# B&R Automation Studio project TD52 (part 148)

### Global_DI.var
```iecst
VAR
	VIS2MM : VIS2MM_DI_struct;
	MM2VIS : MM2VIS_DI_struct;
	Para : Para_DI_struct;
	IN_DI : IN_DI_struct;
	OUT_DI : OUT_DI_struct;
	OPC2MM : OPC2MM_DI_struct;
	bComOpcBitTB : BOOL; (*Kommunikation Bit vom Prüfstand über OPC*)
	TON_bComOpcBitTB : TON; (*AliveTime von Opc-Verbindung*)
	TON_bComOpcFailTB : TON; (*Störung Opc-Verbindung*)
	bComOpcBitMDE : BOOL; (*Kommunikation Bit vom Prüfstand über OPC*)
	TON_bComOpcBitMDE : TON; (*AliveTime von Opc-Verbindung MDE*)
	TON_bComOpcFailMDE : TON; (*Störung Opc-Verbindung MDE*)
	rOpcAG_R : ARRAY[0..40] OF REAL; (*REAL-Var zu TB-Control AuxiliariesGeneral*)
	bOpcAG_R : ARRAY[0..30] OF BOOL; (*BOOL-Var zu TB-Control AuxiliariesGeneral*)
	rOpcCU_R : ARRAY[0..50] OF REAL; (*REAL-Var zu TB-Control Customized*)
	rOpcEX_R : ARRAY[0..30] OF REAL; (*REAL-Var zu TB-Control Exhaust*)
	bOpcEX_R : ARRAY[0..20] OF BOOL; (*BOOL-Var zu TB-Control Exhaust*)
	rOpcGT_R : ARRAY[0..50] OF REAL; (*REAL-Var zu TB-Control Gastrain*)
	bOpcGT_R : ARRAY[0..50] OF BOOL; (*BOOL-Var zu TB-Control Gastrain*)
	rOpcHC_R : ARRAY[0..150] OF REAL; (*REAL-Var zu TB-Control HeatingCooling*)
	bOpcHC_R : ARRAY[0..150] OF BOOL; (*BOOL-Var zu TB-Control HeatingCooling*)
	rOpcME_R : ARRAY[0..10] OF REAL; (*REAL-Var zu TB-Control Measurement*)
	bOpcME_R : ARRAY[0..10] OF BOOL; (*BOOL-Var zu TB-Control Measurement*)
	rOpcVE_R : ARRAY[0..50] OF REAL; (*REAL-Var zu TB-Control Ventilation*)
	bOpcVE_R : ARRAY[0..50] OF BOOL; (*BOOL-Var zu TB-Control Ventilation*)
	bOpcMsg_W : ARRAY[0..799] OF BOOL; (*BOOL-Var von TB-Control Message*)
	rOpcAG_W : ARRAY[0..20] OF REAL; (*REAL-Var von TB-Control AuxiliariesGeneral*)
	bOpcAG_W : ARRAY[0..20] OF BOOL; (*BOOL-Var von TB-Control AuxiliariesGeneral*)
	rOpcCU_W : ARRAY[0..50] OF REAL; (*REAL-Var zu TB-Control Customized*)
	rOpcEX_W : ARRAY[0..30] OF REAL; (*REAL-Var von TB-Control Exhaust*)
	bOpcEX_W : ARRAY[0..20] OF BOOL; (*BOOL-Var von TB-Control Exhaust*)
	rOpcGT_W : ARRAY[0..300] OF REAL; (*REAL-Var von TB-Control Gastrain*)
	bOpcGT_W : ARRAY[0..70] OF BOOL; (*BOOL-Var von TB-Control Gastrain*)
	rOpcHC_W : ARRAY[0..380] OF REAL; (*REAL-Var von TB-Control HeatingCooling*)
	bOpcHC_W : ARRAY[0..300] OF BOOL; (*BOOL-Var von TB-Control HeatingCooling*)
	rOpcME_W : ARRAY[0..50] OF REAL; (*REAL-Var von TB-Control Measurement*)
	bOpcME_W : ARRAY[0..20] OF BOOL; (*BOOL-Var von TB-Control Measurement*)
	rOpcVE_W : ARRAY[0..80] OF REAL; (*REAL-Var von TB-Control Ventilation*)
	bOpcVE_W : ARRAY[0..40] OF BOOL; (*BOOL-Var von TB-Control Ventilation*)
	rOpcMDE_R : ARRAY[0..440] OF REAL; (*REAL-Var zu TB-Control Measurement 10ms*)
	bOpcMDE_R : ARRAY[0..20] OF BOOL; (*BOOL-Var zu TB-Control Measurement 10ms*)
	rOpcMDE_W : ARRAY[0..50] OF REAL; (*REAL-Var von TB-Control Measurement 10ms*)
	bOpcMDE_W : ARRAY[0..40] OF BOOL; (*BOOL-Var von TB-Control Measurement 10ms*)
	rGC_CurrentMonth : REAL; (*GC momentaner Monat*)
	rGC_CurrentDay : REAL; (*GC momentaner Tag*)
	rGC_CurrentYear : REAL; (*GC momentanes Jahr*)
	rGC_CurrentHour : REAL; (*GC momentane Stunde*)
	rGC_CurrentMinute : REAL; (*GC momentane Minute*)
	rGC_SampleMonth : REAL; (*GC Probe gezogen Monat*)
	rGC_SampleDay : REAL; (*GC Probe gezogen Tag*)
	rGC_SampleYear : REAL; (*GC Probe gezogen Jahr*)
	rGC_SampleHour : REAL; (*GC Probe gezogen Stunde*)
	rGC_SampleMinute : REAL; (*GC Probe gezogen Minute*)
	TON_DemDataMan_GC : TON; (*Damit der Visu-Button wieder auf FALSE geschrieben wird*)
	rEndurTestTimeMinute : REAL; (*Dauerlauf beendet Tagesminute*)
	rEndurTestTimeHour : REAL; (*Dauerlauf beendet Tagesstunde*)
	rEndurTestTimeDay : REAL; (*Dauerlauf beendet Tag vom Monat*)
	rEndurTestTimeWDay : REAL; (*Dauerlauf beendet Wochentag*)
	rEndurTestTimeMonth : REAL; (*Dauerlauf beendet Monat*)
	rEndurTestTimeYear : REAL; (*Dauerlauf beendet Jahr*)
	rP_MDE_OPC_Set : REAL; (*Externe Leistungsvorgabe von Messtechnik*)
	bMDEBusAlive : BOOL; (*Bus-Verbindung vorhanden für Leistungsvorgabe von Messtechnik*)
	bMDEOPC_Dem : BOOL; (*Anforderung externe Leistungsvorgabe von Messtechnik*)
	RS_Ctr_ChCW_LT : RS; (*Aktivierung Y_Set für Offset*)
	RS_Ctr_ChCW_HT : RS; (*Aktivierung Y_Set für Offset*)
	RS_Ctr_ChCW_LT_LP : RS; (*Aktivierung Y_Set für Offset*)
	RS_Ctr_ChCW_LT_HP : RS; (*Aktivierung Y_Set für Offset*)
	RS_Ctr_ChCW_HT_LP : RS; (*Aktivierung Y_Set für Offset*)
	RS_Ctr_ChCW_HT_HP : RS; (*Aktivierung Y_Set für Offset*)
	RS_Ctr_ECW : RS; (*Aktivierung Y_Set für Offset*)
	RS_Ctr_OCW : RS; (*Aktivierung Y_Set für Offset*)
	bCtr_LT_In_Y_set_Active : BOOL; (*Y_Set für Offset aktiv*)
	bCtr_HT_In_Y_set_Active : BOOL; (*Y_Set für Offset aktiv*)
	bCtr_LT_LP_In_Y_set_Active : BOOL; (*Y_Set für Offset aktiv*)
	bCtr_LT_HP_In_Y_set_Active : BOOL; (*Y_Set für Offset aktiv*)
	bCtr_HT_LP_In_Y_set_Active : BOOL; (*Y_Set für Offset aktiv*)
	bCtr_HT_HP_In_Y_set_Active : BOOL; (*Y_Set für Offset aktiv*)
	bCtr_ECW_In_Y_set_Active : BOOL; (*Y_Set für Offset aktiv*)
	bCtr_OCW_In_Y_set_Active : BOOL; (*Y_Set für Offset aktiv*)
	bBlock_MG_TB : BOOL; (*Block mixgas controller from TB CPU*)
	bBlock_SG_TB : BOOL; (*Block special gas from TB CPU*)
	bDem_GT3 : BOOL; (*activation bit for custom gastrain 3*)
	rGT_RatioAdd : REAL; (*add mixing setpoint for custom gastrain 3*)
	rH2_Set : REAL; (*setpoint addmixing H2*)
	rH2_Act_Calc : REAL; (*Actual volume H2 content calculated (gas meter)*)
	rH2_Act_Cube : REAL; (*Actual volume H2 content measurement cube*)
	rTB_Version : REAL; (*Gesendete Version von TB_Control*)
	bPreHeatWDayLT_On : BOOL; (*Einschalten der Vorwärmung über Zeitsteuerung*)
	usDurationPI_A : UINT := 0; (*PI Duration Bank A*)
	usDurationPI_B : UINT := 0; (*PI Duration Bank B*)
END_VAR
```

### Data object Logical/DataInterface/META_DI (Simple) - Simple data object.

#### META_DI.dat
```
; *******************************************************************************
; AGGR: Module Meta Data (data module)
;
; This code is confidential and proprietary to the INNIO Company.
; It may not be used in any form, or reproduced in any manner, without the express
; written permission of the INNIO Company.
; Copyright, INNIO Company, 2022
;
; Customized modifications: -
; ------------------------
;
; History:
; -------
; V1.00.0	14.11.2022	Vockenberger	Neu erstellt
;
; Instructions for use:
; --------------------
; make only changes at the version numbers
;
; Outstandings:
; ------------
;
; *******************************************************************************
;
"<META>"
;
; Module ID
"<MODUL>DI</MODUL>"
;
; Module Version (xx.yy.zz.cc)
"<VERSION>01.01.00.00</VERSION>"
;
; Module Basisupdate Version BU (00-99)
"<BASISUPDATE_VERSION>00</BASISUPDATE_VERSION>"
;
; Optional: specify order number for limitated module usage
"<ORDER></ORDER>" ;<!--(optional for restricted customizations; missing statement makes module valid for all orders)-->
;
; Permanent Datamodule Filenames<!-- NAME ist ohne Dateiendung einzutragen; Nur für Counter und interne Parameter verwenden-->
"<DATAMODULES>" ;<!-- optional; mehrere DATAMODULES erlaubt-->
"	<DATAMODULE>perm_DI</DATAMODULE>"
"	<DATAMODULE>VISpm_DI</DATAMODULE>"
"</DATAMODULES>"
;
"</META>"
```

### Program Logical/DataInterface/Gnl_AG (IEC) - General Var edit

#### Gnl_AG.st
```iecst
(*******************************************************************************
Gnl_AG		Allgemeine Verarbeitung von Variablen

This code is confidential AND proprietary to the INNIO Company.
It may NOT be used in any form, or reproduced in any manner, without the express
written permission of the INNIO Company.
Copyright, INNIO Company, 2022

Customized modifications: -
------------------------

History:
-------
V1.00.0	14.09.2022		Vockenberger	Neu erstellt
V1.01.0	31.05.2023		Vockenberger	Gaskompressor mit Parameterabfrage und Betriebsstundenzähler mit Wartungsanforderung
										Dauerlauftest
		11.07.2023		Gruber St.		Hinzugefügt: Gasventil 3, Parameter & Anzeigen Gastrain, diverse Abfragen für Visu
		31.07.2023		Vockenberger	Struktur von General_DI geändert
V1.02.0 20.03.2024		Vockenberger	Parameter für Visu Aktivierungen hinzugefügt
		11.04.2024		Vockenberger	Version von 1.01.0 auf 1.02.0 erhöht
V1.02.1 16.10.2024		Vockenberger	Version 1.02.1
V1.03.0	09.01.2025		Gruber St.		cleanUp after change of parameter structure

Instructions FOR use:
--------------------

Outstandings:
------------

*******************************************************************************)

PROGRAM _CYCLIC

	(*DataInterface Version auf Visu Übertragen*)
	MM2VIS.stDI_Version := '1.03.5';

	(*TB_Control Version auf Visu Übertragen*)
	stTB_Version := REAL_TO_STRING(rTB_Version);
	stTB_VersionConfig1 := INSERT(stTB_Version, '.', 1);
	stTB_VersionConfig2 := INSERT(stTB_VersionConfig1, '.', 4);
	strcpy( ADR(MM2VIS.stTB_Version), ADR(stTB_VersionConfig2) );

	(* Parameter für Visu Aktivierungen *)
	Para.bExtCtrNOX_Active;

	(* Zeitsteuerung von Vorwärmung wird Deaktiverit *)
	FOR i:= 0 TO 6 DO
		IF VIS2MM.bECW_PreH_Dem_Customized THEN (*Wenn die Vorwärmung auf der Visu deaktiviert wird, wird die Zeitsteurung auch unterbrochen, bis zum nächsten aktivierten Tag*)
			Para.tPreHeatWDay[i].Off := TRUE;
		ELSE
			Para.tPreHeatWDay[i].Off := FALSE;
		END_IF
	END_FOR

	(* Oil level umrechnen auf % damit der Tank die Füllmenge richtig anzeigt *)
	IF MM2VIS.rLevel_Oiltank > Para.rLevel_Oiltank_ScalY1 AND (Para.rLevel_Oiltank_ScalY2 > 0.0) THEN
		MM2VIS.rLevel_OilNorm := MM2VIS.rLevel_Oiltank/Para.rLevel_Oiltank_ScalY2 *100;
	ELSE
		MM2VIS.rLevel_OilNorm := 0;
	END_IF

	(* Dauerlauftest *)
	DT_EndurTest.minute := REAL_TO_USINT(rEndurTestTimeMinute);
	DT_EndurTest.hour := REAL_TO_USINT(rEndurTestTimeHour);
	DT_EndurTest.day := REAL_TO_USINT(rEndurTestTimeDay);
	DT_EndurTest.wday := REAL_TO_USINT(rEndurTestTimeWDay);
	DT_EndurTest.month := REAL_TO_USINT(rEndurTestTimeMonth);
	DT_EndurTest.year := REAL_TO_UINT(rEndurTestTimeYear);

	ascDTStructure(ADR(DT_EndurTest),ADR(stEndurTestAll),25);
	stFind := ':'; //Es wird nach : gesucht
	iPosition := FIND(stEndurTestAll, stFind);
	szResultString := DELETE(stEndurTestAll, 15, iPosition+3); //Wenn : gefunden wurde, die Position + 3 damit die Position, ab der gelöscht werden soll bestimmt wird
	szDateString := LEFT(szResultString, 10);
	szTimeString := RIGHT(szResultString, 5);

	strcpy( ADR(MM2VIS.stEndurTestDate), ADR(szDateString) );
	strcpy( ADR(MM2VIS.stEndurTestTime), ADR(szTimeString) );

	IF EDGEPOS(MM2VIS.bEndurTestEnd) THEN
		VIS2MM.bEndurTestStart := FALSE; //Start Schalter wird auf False geschrieben, wenn der Test beendet ist
	END_IF

	(*Visu-Button Lüftung auf Automatik wird bei Anfoderung HBT auf TRUE geschrieben*)
	IF IN_DI.bEng_Run OR EDGEPOS(IN_DI.bEng_Aux_Dem_CDR) THEN
		VIS2MM.bDem_ERV_Aut_Vis := TRUE;
	END_IF

	(*Service Page Variablen, nur vorbereitet, keine Funktion*)
	VIS2MM.bManCircLouActive;
	VIS2MM.bManCircLouEngActive;
	VIS2MM.bManDem_PCG_Val;
	VIS2MM.bManFV_PCGC_MG;
	VIS2MM.bManGV_Active;
	VIS2MM.bManGV_NG_Set;
	VIS2MM.bManGV_PG_Set;
	VIS2MM.bManGV_SG_Set;
	VIS2MM.bManInAirFanActive;
	VIS2MM.bManInEngAirFanActive;
	VIS2MM.bManInlLouActive;
	VIS2MM.bManInlLouEngActive;
	VIS2MM.bManInlLouRoomActive;
	VIS2MM.bManOutAirFanActive;
	VIS2MM.bManOutlLouActive;
	VIS2MM.bManPCG_Comp_Active;
	VIS2MM.bManPCG_DemCoolFan;
	VIS2MM.bManPCG_DemReliefValve;
	VIS2MM.bManPCG_DemValCW;
	VIS2MM.bManPCG_GC_Dem;
	VIS2MM.bManPCG_GV_MG_Set;
	VIS2MM.bManPCG_GV_NG_Set;
	VIS2MM.bManPCG_GV_PG_Set;
	VIS2MM.rManCircLouEngSet;
	VIS2MM.rManCircLouSet;
	VIS2MM.rManInAirFanSet;
	VIS2MM.rManInEngAirFanSet;
	VIS2MM.rManInlLouEngSet;
	VIS2MM.rManInlLouRoomSet;
	VIS2MM.rManInlLouSet;
	VIS2MM.rManOutAirFanSet;
	VIS2MM.rManOutlLouSet;

END_PROGRAM
```

#### Gnl_AG.var
```iecst
VAR
	i : INT;
	DT_EndurTest : DTStructure; (*Date and Time Struktur zu weiter Verarbeitung*)
	stFind : STRING[10]; (*Das was im String gesucht wird*)
	stEndurTestAll : STRING[25]; (*Dauerlauftest Datum ganzer String*)
	iPosition : INT; (*Position von : im String*)
	szResultString : STRING[25]; (*Bearbeiteter String*)
	szDateString : STRING[11]; (*Bearbeiteter String, der auf die Visu geschrieben werden kann*)
	szTimeString : STRING[6]; (*Bearbeiteter String, der auf die Visu geschrieben werden kann*)
	stTB_Version : STRING[10]; (*Versionsanzeige TB_Control von REAL auf STRING umgewandelt*)
	stTB_VersionConfig1 : STRING[10]; (*Für TB_Control Versionsanzeige wird der reste Punkt eingefügt*)
	stTB_VersionConfig2 : STRING[6]; (*Für TB_Control Versionsanzeige wird der zweite Punkt eingefügt*)
END_VAR
```

### Program Logical/DataInterface/Gnl_GT (IEC) - General Var edit

#### Gnl_GT.st
```iecst
(*******************************************************************************
Gnl_GT		Allgemeine Verarbeitung von Variablen

This code is confidential AND proprietary to the INNIO Company.
It may NOT be used in any form, or reproduced in any manner, without the express
written permission of the INNIO Company.
Copyright, INNIO Company, 2022

- list addidtional customized IO channels

Customized modifications: -
------------------------

History:
-------
V1.00.0	14.09.2022		Vockenberger	Neu erstellt
V1.01.0	31.05.2023		Vockenberger	Gaskompressor mit Parameterabfrage und Betriebsstundenzähler mit Wartungsanforderung
										Dauerlauftest
										Externe Leistungsvorgabe, umschaltung von Prüfstand/PUMA auf EnergyManagement
		11.07.2023		Gruber St.		Hinzugefügt: Gasventil 3, Parameter & Anzeigen Gastrain, diverse Abfragen für Visu
		31.07.2023		Vockenberger	Struktur von General_DI geändert
		09.01.2024		Gruber St.		added blockage bits for mixgas & special gas
V1.01.1	19.03.2024		Gruber St.		added vis mixgas ratio from IN_DI
		27.03.2024		Gruber St.		added vis H2 measurement cube
V1.02.0	22.04.2024		Gruber St.		Parameter for several vis; MFC open vis
V1.03.0	14.01.2025		Gruber St.		several changes for new para struct

Instructions FOR use:
--------------------

Outstandings:
------------

*******************************************************************************)

PROGRAM _CYCLIC

	(* ----------------------------------------------------------------------------*)
	(*Uhrzeit vom GC generieren*)
	iGC_CurrentDay := REAL_TO_SINT(rGC_CurrentDay);
	iGC_CurrentMonth := REAL_TO_USINT(rGC_CurrentMonth);
	iGC_CurrentYear := REAL_TO_UINT(rGC_CurrentYear);
	iGC_CurrentHour := REAL_TO_USINT(rGC_CurrentHour);
	iGC_CurrentMinute := REAL_TO_USINT(rGC_CurrentMinute);

	iGC_SampleDay := REAL_TO_SINT(rGC_SampleDay);
	iGC_SampleMonth := REAL_TO_USINT(rGC_SampleMonth);
	iGC_SampleYear := REAL_TO_UINT(rGC_SampleYear);
	iGC_SampleHour := REAL_TO_USINT(rGC_SampleHour);
	iGC_SampleMinute := REAL_TO_USINT(rGC_SampleMinute);

	GC_CurrentDate.day := iGC_CurrentDay;
	GC_CurrentDate.month := iGC_CurrentMonth;
	GC_CurrentDate.year := iGC_CurrentYear;

	GC_CurrentTIME.hour := iGC_CurrentHour;
	GC_CurrentTIME.minute := iGC_CurrentMinute;

	GC_SampleDate.day := iGC_SampleDay;
	GC_SampleDate.month := iGC_SampleMonth;
	GC_SampleDate.year := iGC_SampleYear;

	GC_SampleTIME.hour := iGC_SampleHour;
	GC_SampleTIME.minute := iGC_SampleMinute;

	LenTime:=6;
	LenDate:=25;
	ascDTStructure(ADR(GC_CurrentDate),ADR(MM2VIS.stGC_CurrentDate),LenDate);  (* converts TIMEStructure to a string *)
	ascTIMEStructure(ADR(GC_CurrentTIME),ADR(MM2VIS.stGC_CurrentTIME),LenTime);

	ascDTStructure(ADR(GC_SampleDate),ADR(MM2VIS.stGC_SampleDate),LenDate);
	ascTIMEStructure(ADR(GC_SampleTIME),ADR(MM2VIS.stGC_SampleTIME),LenTime);

	(* ----------------------------------------------------------------------------*)
	(* Visualization mixgas ratio *)
	IF Para.bGasFlowCtr AND NOT Para.bIncl_SG_Calc OR (NOT Para.bGasFlowCtr AND NOT Para.bIncl_SG_Calc) THEN
		MM2VIS.rVol_NG_PG := MM2VIS.rVol_NG + MM2VIS.rVol_PG - MM2VIS.rVol_SG;
	ELSE
		MM2VIS.rVol_NG_PG := MM2VIS.rVol_NG + MM2VIS.rVol_PG; (* part of special gas already included *)
	END_IF;

	(* Visualization MFC propan gas open *)
	IF MM2VIS.rCtr_MFC_PG > 0.01 THEN
		MM2VIS.bMFC_PG_open_vis := TRUE;
	ELSE
		MM2VIS.bMFC_PG_open_vis := FALSE;
	END_IF;

	(* Visualization MFC special gas open *)
	IF MM2VIS.rCtr_MFC_SG > 0.01 THEN
		MM2VIS.bMFC_SG_open_vis := TRUE;
	ELSE
		MM2VIS.bMFC_SG_open_vis := FALSE;
	END_IF;

	(* Visualization H2 measurement cube *)
	MM2VIS.rH2_Act_Cube	:= rH2_Act_Cube * 100;

	(* Abfrage für Freigabe Mischgas-Regler mittels Gasdosierventil - Gas 1-2/3 *)
	IF IN_DI.iIdx_Gastyp = 3
		AND IN_DI.iNum_GT = 2
		AND IN_DI.bTJ_Exist = TRUE
		AND IN_DI.iN_GMU_Devices > 1
		AND IN_DI.bGT_MixActive = TRUE
		AND (IN_DI.iIdx_SelGasTyp = 6 OR IN_DI.iIdx_SelGasTyp = 5)
		AND MM2VIS.bDem_GV_PG
		AND NOT MM2VIS.bDem_GV_SG THEN
		MM2VIS.bParaGasMixEngOk := TRUE;
	ELSE
		MM2VIS.bParaGasMixEngOk := FALSE;
	END_IF;

	(* Abfrage für Freigabe Mischgas-Regler mittels MFC - Gas 1-2 *)
	IF IN_DI.iIdx_Gastyp >= 2
		AND IN_DI.iIdx_SelGasTyp = 0
		AND IN_DI.bGT_CVActive
		AND IN_DI.bGT_CVIpol12Active THEN
		MM2VIS.bParaGasMixMFCOk := TRUE;
	ELSE
		MM2VIS.bParaGasMixMFCOk := FALSE;
	END_IF

	(* Freigabe Mischgas für Anzeige auf Visu *)
	IF MM2VIS.bParaGasMixMFCOk OR MM2VIS.bParaGasMixEngOk THEN
		MM2VIS.bRelMixGas := TRUE;
	ELSE
		MM2VIS.bRelMixGas := FALSE;
	END_IF;

	(* Switch Mixgas from MN-Controller to Volume - Gas 1-2 *)
	IF EDGENEG(MM2VIS.bParaGasMixMFCOk AND NOT (MM2VIS.bDem_GV_NG AND MM2VIS.bDem_GV_PG AND MM2VIS.bDem_GV_SG AND Para.bIncl_SG_Calc)) AND VIS2MM.bCtr_MN_MG_active THEN
		VIS2MM.bVolPG_Man := TRUE;
	END_IF;

	(* Switch Mixgas from MN-Controller to Off - Gas 1-2/3 *)
	IF EDGENEG(MM2VIS.bParaGasMixEngOk AND NOT (MM2VIS.bDem_GV_NG AND MM2VIS.bDem_GV_PG AND MM2VIS.bDem_GV_SG AND Para.bIncl_SG_Calc)) AND VIS2MM.bCtr_MN_MG_active THEN
		VIS2MM.bCtr_MN_MG_off := TRUE;
	END_IF;

	(* Block mixgas controller *)
	IF bBlock_MG_TB OR MM2VIS.bMsg7000 THEN
		VIS2MM.bCtr_MN_MG_off := TRUE;
	END_IF;

	(* Block specialgas mixing *)
	IF bBlock_SG_TB OR MM2VIS.bMsg7000 THEN
		VIS2MM.rVol_SG_Set := 0;
	END_IF;

	(* Externe Anforderung MZ von PUMA *)
	IF VIS2MM.bExtMN_ActiveMDE AND MM2VIS.bExtMNFromMDE THEN
		VIS2MM.bCtr_MN_MG_active := TRUE;
		Para.tCtr_MN_MG.W_set := MM2VIS.rExtMN_Set;
	END_IF;

	IF EDGENEG(VIS2MM.bExtMN_ActiveMDE) THEN
		VIS2MM.bCtr_MN_MG_off := TRUE;
	END_IF;

	(* Switch Mixgas from Volume to OFF *)
	IF EDGENEG(MM2VIS.bParaGasMixMFCOk OR (MM2VIS.bDem_GV_NG AND MM2VIS.bDem_GV_PG AND MM2VIS.bDem_GV_SG)) AND VIS2MM.bVolPG_Man THEN
		VIS2MM.bCtr_MN_MG_off := TRUE;
	END_IF;

	(* Wenn MN Bechrechnung inaktiv, dann wird der MN-Regler deaktiviert *)
	IF EDGENEG(MM2VIS.bMN_Cal_Status) THEN
		VIS2MM.bCtr_MN_MG_off := TRUE;
	END_IF;

	(* MN Ctr from MN to OFF *)
	IF EDGEPOS(VIS2MM.bCtr_MN_MG_off) AND VIS2MM.bCtr_MN_MG_active THEN
		Para.tCtr_MN_MG.W_set := 100;
	ELSE
		Para.tCtr_MN_MG.W_set := Para.tCtr_MN_MG.W_set;
	END_IF

	(* MN Ctr from Volume to OFF *)
	IF EDGEPOS(VIS2MM.bCtr_MN_MG_off) AND VIS2MM.bVolPG_Man THEN
		VIS2MM.rVol_PG_Set := 0;
	ELSE
		VIS2MM.rVol_PG_Set := VIS2MM.rVol_PG_Set;
	END_IF

	(* MN Ctr from MN to VOL *)
	IF EDGEPOS(VIS2MM.bVolPG_Man) AND VIS2MM.bCtr_MN_MG_active THEN
		VIS2MM.rVol_PG_Set := MM2VIS.rVol_PG;
	ELSE
		VIS2MM.rVol_PG_Set := VIS2MM.rVol_PG_Set;
	END_IF

	(* MN Ctr from VOL to MN *)
	IF EDGEPOS(VIS2MM.bCtr_MN_MG_active) AND VIS2MM.bVolPG_Man THEN
		Para.tCtr_MN_MG.W_set := MM2VIS.rMN_MG;
	ELSE
		Para.tCtr_MN_MG.W_set := Para.tCtr_MN_MG.W_set;
	END_IF

	(* Regler Methane Button Steuerung *)
	 IF EDGEPOS(VIS2MM.bCtr_MN_MG_active) THEN
		VIS2MM.bCtr_MN_MG_off := FALSE;
		VIS2MM.bVolPG_Man := FALSE;
	ELSE
		VIS2MM.bCtr_MN_MG_off := VIS2MM.bCtr_MN_MG_off;
		VIS2MM.bVolPG_Man := VIS2MM.bVolPG_Man;
	END_IF

	IF EDGEPOS(VIS2MM.bCtr_MN_MG_off) THEN
		VIS2MM.bCtr_MN_MG_active := FALSE;
		VIS2MM.bVolPG_Man := FALSE;
	ELSE
		VIS2MM.bCtr_MN_MG_active := VIS2MM.bCtr_MN_MG_active;
		VIS2MM.bVolPG_Man := VIS2MM.bVolPG_Man;
	END_IF

	IF EDGEPOS(VIS2MM.bVolPG_Man) THEN
		VIS2MM.bCtr_MN_MG_active := FALSE;
		VIS2MM.bCtr_MN_MG_off := FALSE;
	ELSE
		VIS2MM.bCtr_MN_MG_active := VIS2MM.bCtr_MN_MG_active;
		VIS2MM.bCtr_MN_MG_off := VIS2MM.bCtr_MN_MG_off;
	END_IF

	IF EDGENEG(MM2VIS.bDem_GV_SG) THEN
		VIS2MM.rVol_SG_Set := 0;
	ELSE
		VIS2MM.rVol_SG_Set := VIS2MM.rVol_SG_Set;
	END_IF

	(* ----------------------------------------------------------------------------*)
	(* Gaskompressor Wartungsanforderung *)
	IF Para.bGasCompActive THEN
		xComp_OpHour(enable := MM2VIS.bPr_PCG_GC_Dem, BH_adr := ADR(ComOpHour_Imp.tick));
		xTOF_CompOpHour(IN := xComp_OpHour.BH_Imp, PT := T#10s);
		IF EDGEPOS(xTOF_CompOpHour.Q) THEN
			Para.rCnt_CompOpHoursW := Para.rCnt_CompOpHoursW - 1;					(* increase counter *)
		END_IF
		Para.rCnt_CompOpHoursW 			:= Para.rCnt_CompOpHoursW;

		IF Para.rCnt_CompOpHoursW <= 0 THEN
			OUT_DI.bCompOpHoursWarning := TRUE;
		ELSE
			OUT_DI.bCompOpHoursWarning := FALSE;
		END_IF
	END_IF

	(* ----------------------------------------------------------------------------*)
	(* set PG trace heating on, with time control *)
	IF EDGEPOS(MM2VIS.bPG_TraceHeat_TimeCtr_On) THEN
		VIS2MM.bSel_PG_TraceHeat := TRUE;
	END_IF

	(* ----------------------------------------------------------------------------*)
	(* Added Parameter bSA_PI_Active AND to TB_Control-VIS *)
	MM2VIS.bSA_PI_Active := IN_DI.bSA_PI_Active;
	MM2VIS.rCA_PI_Dur_Avg := IN_DI.rCA_PI_Dur_Avg;

END_PROGRAM
```

#### Gnl_GT.var
```iecst
VAR
	iGC_CurrentDay : USINT; (*GC momentaner Tag*)
	iGC_CurrentMonth : USINT; (*GC momentaner Monat*)
	iGC_CurrentYear : UINT; (*GC momentanes Jahr*)
	iGC_CurrentHour : USINT; (*GC momentane Stunde*)
	iGC_CurrentMinute : USINT; (*GC momentane Minute*)
	iGC_SampleDay : USINT; (*GC Probe gezogen Tag*)
	iGC_SampleMonth : USINT; (*GC Probe gezogen Monat*)
	iGC_SampleYear : UINT; (*GC Probe gezogen Jahr*)
	iGC_SampleHour : USINT; (*GC Probe gezogen Stunde*)
	iGC_SampleMinute : USINT; (*GC Probe gezogen Minute*)
	GC_SampleTIME : TIMEStructure; (*GC TimeStructure für VisuString*)
	GC_CurrentTIME : TIMEStructure; (*GC TimeStructure für VisuString*)
	GC_SampleDate : DTStructure; (*GC DateStructure für VisuString*)
	GC_CurrentDate : DTStructure; (*GC DateStructure für VisuString*)
	LenTime : UDINT; (*GC VisuString-Länge für Anzeige*)
	LenDate : UDINT; (*GC VisuString-Länge für Anzeige*)
	ComOpHour_Imp : bh_typ; (*Compressor operation hours counter*)
	xComp_OpHour : BH; (*Hour counter for compressor operating hours*)
	xTOF_CompOpHour : TOF; (*Off delay for compressor operating hours*)
END_VAR
```

### Program Logical/DataInterface/Gnl_HC (IEC) - General Var edit

#### Gnl_HC.st
```iecst
(*******************************************************************************
Gnl_HC		Allgemeine Verarbeitung von Variablen

This code is confidential AND proprietary to the INNIO Company.
It may NOT be used in any form, or reproduced in any manner, without the express
written permission of the INNIO Company.
Copyright, INNIO Company, 2023

- list addidtional customized IO channels

Customized modifications: -
------------------------

History:
-------
V1.01.0	27.05.2023		Vockenberger	Manuelle Anforderung der Kühlkreispumpen, wenn BWS auf Aus ist.
		31.07.2023		Vockenberger	Struktur von General_DI geändert
		09.10.2023		Vockenberger	Offset für Kühlkreis-Regelventile bei Eng_Run eingefügt

Instructions FOR use:
--------------------

Outstandings:
------------

*******************************************************************************)

PROGRAM _CYCLIC

	(* Manuelle Anforderung der Kühlwasserpumpen, wenn Betriebswahlschalter auf aus ist *)
	MM2VIS.iIdx_OMSS := IN_DI.iIdx_OMSS;	//Damit auf der Visualisierung die Schalter verreigelt werden können
	IF IN_DI.iIdx_OMSS = 0 AND NOT IN_DI.bEng_Aux_Dem_CDR THEN
		VIS2MM.bMan_ECW_Pump;
		VIS2MM.bMan_OCW_Pump;
		VIS2MM.bMan_LT_Pump;
		VIS2MM.bMan_HT_Pump;
		VIS2MM.bMan_LT_LP_Pump;
		VIS2MM.bMan_LT_HP_Pump;
		VIS2MM.bMan_HT_LP_Pump;
		VIS2MM.bMan_HT_HP_Pump;
	ELSE
		VIS2MM.bMan_ECW_Pump := FALSE;
		VIS2MM.bMan_OCW_Pump := FALSE;
		VIS2MM.bMan_LT_Pump := FALSE;
		VIS2MM.bMan_HT_Pump := FALSE;
		VIS2MM.bMan_LT_LP_Pump := FALSE;
		VIS2MM.bMan_LT_HP_Pump := FALSE;
		VIS2MM.bMan_HT_LP_Pump := FALSE;
		VIS2MM.bMan_HT_HP_Pump := FALSE;
	END_IF

	(*Aktivierung Offset für Kühlkreis-Regelventile bei Eng_Run*)
	RS_Ctr_ChCW_LT(SET:=EDGEPOS(IN_DI.bEng_Run), RESET1:=(VIS2MM.tCtr_ChCW_LT_In.Y_set < MM2VIS.tCtr_ChCW_LT_Out.Y) OR (EDGENEG(IN_DI.bEng_Run)));
	IF VIS2MM.tCtr_ChCW_LT_In.Y_set_Active AND RS_Ctr_ChCW_LT.Q1 THEN
		bCtr_LT_In_Y_set_Active :=  TRUE;
	ELSE
		bCtr_LT_In_Y_set_Active :=  FALSE;
	END_IF

	RS_Ctr_ChCW_HT(SET:=EDGEPOS(IN_DI.bEng_Run), RESET1:=(VIS2MM.tCtr_ChCW_HT_In.Y_set < MM2VIS.tCtr_ChCW_HT_Out.Y) OR (EDGENEG(IN_DI.bEng_Run)));
	IF VIS2MM.tCtr_ChCW_HT_In.Y_set_Active AND RS_Ctr_ChCW_HT.Q1 THEN
		bCtr_HT_In_Y_set_Active :=  TRUE;
	ELSE
		bCtr_HT_In_Y_set_Active :=  FALSE;
	END_IF

	RS_Ctr_ChCW_LT_LP(SET:=EDGEPOS(IN_DI.bEng_Run), RESET1:=(VIS2MM.tCtr_ChCW_LT_LP_In.Y_set < MM2VIS.tCtr_ChCW_LT_LP_Out.Y) OR (EDGENEG(IN_DI.bEng_Run)));
	IF VIS2MM.tCtr_ChCW_LT_LP_In.Y_set_Active AND RS_Ctr_ChCW_LT_LP.Q1 THEN
		bCtr_LT_LP_In_Y_set_Active :=  TRUE;
	ELSE
		bCtr_LT_LP_In_Y_set_Active :=  FALSE;
	END_IF

	RS_Ctr_ChCW_LT_HP(SET:=EDGEPOS(IN_DI.bEng_Run), RESET1:=(VIS2MM.tCtr_ChCW_LT_HP_In.Y_set < MM2VIS.tCtr_ChCW_LT_HP_Out.Y) OR (EDGENEG(IN_DI.bEng_Run)));
	IF VIS2MM.tCtr_ChCW_LT_HP_In.Y_set_Active AND RS_Ctr_ChCW_LT_HP.Q1 THEN
		bCtr_LT_HP_In_Y_set_Active :=  TRUE;
	ELSE
		bCtr_LT_HP_In_Y_set_Active :=  FALSE;
	END_IF

	RS_Ctr_ChCW_HT_LP(SET:=EDGEPOS(IN_DI.bEng_Run), RESET1:=(VIS2MM.tCtr_ChCW_HT_LP_In.Y_set < MM2VIS.tCtr_ChCW_HT_LP_Out.Y) OR (EDGENEG(IN_DI.bEng_Run)));
	IF VIS2MM.tCtr_ChCW_HT_LP_In.Y_set_Active AND RS_Ctr_ChCW_HT_LP.Q1 THEN
		bCtr_HT_LP_In_Y_set_Active :=  TRUE;
	ELSE
		bCtr_HT_LP_In_Y_set_Active :=  FALSE;
	END_IF

	RS_Ctr_ChCW_HT_HP(SET:=EDGEPOS(IN_DI.bEng_Run), RESET1:=(VIS2MM.tCtr_ChCW_HT_HP_In.Y_set < MM2VIS.tCtr_ChCW_HT_HP_Out.Y) OR (EDGENEG(IN_DI.bEng_Run)));
	IF VIS2MM.tCtr_ChCW_HT_HP_In.Y_set_Active AND RS_Ctr_ChCW_HT_HP.Q1 THEN
		bCtr_HT_HP_In_Y_set_Active :=  TRUE;
	ELSE
		bCtr_HT_HP_In_Y_set_Active :=  FALSE;
	END_IF

	RS_Ctr_ECW(SET:=EDGEPOS(IN_DI.bEng_Run), RESET1:=(VIS2MM.tCtr_ECW_In.Y_set < MM2VIS.tCtr_ECW_Out.Y) OR (EDGENEG(IN_DI.bEng_Run)));
	IF VIS2MM.tCtr_ECW_In.Y_set_Active AND RS_Ctr_ECW.Q1 THEN
		bCtr_ECW_In_Y_set_Active :=  TRUE;
	ELSE
		bCtr_ECW_In_Y_set_Active :=  FALSE;
	END_IF

	RS_Ctr_OCW(SET:=EDGEPOS(IN_DI.bEng_Run), RESET1:=(VIS2MM.tCtr_OCW_In.Y_set < MM2VIS.tCtr_OCW_Out.Y) OR (EDGENEG(IN_DI.bEng_Run)));
	IF VIS2MM.tCtr_OCW_In.Y_set_Active AND RS_Ctr_ECW.Q1 THEN
		bCtr_OCW_In_Y_set_Active :=  TRUE;
	ELSE
		bCtr_OCW_In_Y_set_Active :=  FALSE;
	END_IF

	(*Aktivierung NT Vorwärmung, wenn Betriebswahlschalter auf aus ist über Zeitsteuerung*)
	IF EDGEPOS(bPreHeatWDayLT_On) THEN	(*Aktivierung Vorwärmung vom Prüfstand über eine positiven Flanke*)
		VIS2MM.bLT_PreH_Dem := TRUE;
	ELSE
		VIS2MM.bLT_PreH_Dem := VIS2MM.bLT_PreH_Dem;
	END_IF

	(* Zeitsteuerung von NT Vorwärmung wird Deaktiverit *)
	FOR i:= 0 TO 6 DO
		IF VIS2MM.bLT_PreH_Dem THEN (*Wenn die Vorwärmung auf der Visu deaktiviert wird, wird die Zeitsteurung auch unterbrochen, bis zum nächsten aktivierten Tag*)
			VIS2MM.tPreHeatWDayLT[i].Off := TRUE;
		ELSE
			VIS2MM.tPreHeatWDayLT[i].Off := FALSE;
		END_IF
	END_FOR

END_PROGRAM
```

#### Gnl_HC.var
```iecst
VAR
	i : INT;
END_VAR
```

### Program Logical/DataInterface/Gnl_ME (IEC) - General Var edit

#### Gnl_ME.st
```iecst
(*******************************************************************************
Gnl_ME		Allgemeine Verarbeitung von Variablen

This code is confidential AND proprietary to the INNIO Company.
It may NOT be used in any form, or reproduced in any manner, without the express
written permission of the INNIO Company.
Copyright, INNIO Company, 2023

- list addidtional customized IO channels

Customized modifications: -
------------------------

History:
-------
V1.01.0	31.05.2023	Vockenberger	Externe Leistungsvorgabe, umschaltung von Prüfstand/PUMA auf EnergyManagement
		31.07.2023	Vockenberger	Struktur von General_DI geändert
V1.03.0 10.06.2025	Vockenberger	added extern setpoint for CAT temp over MDE

Instructions FOR use:
--------------------

Outstandings:
------------

*******************************************************************************)

PROGRAM _CYCLIC

	(* Externe Leistungsvorgabe, umschaltung von Prüfstand/PUMA auf EnergyManagement *)
	IF VIS2MM.iSelExtP_OPC_Set = 0 THEN //Externe Leistungvorgabe deaktiviert
		MM2VIS.rP_OPC_Set;
		MM2VIS.bBusAlive := bMDEBusAlive;
		MM2VIS.bOPC_Dem := FALSE;
	ELSIF VIS2MM.iSelExtP_OPC_Set = 1 THEN //Externe Leistungvorgabe über MDE
		MM2VIS.rP_OPC_Set	:= rP_MDE_OPC_Set;
		MM2VIS.bBusAlive := bMDEBusAlive;
		MM2VIS.bOPC_Dem := bMDEOPC_Dem;
	ELSIF VIS2MM.iSelExtP_OPC_Set = 2 THEN  //Externe Leistungvorgabe über EnergyManagement
		MM2VIS.rP_OPC_Set := OPC2MM.rP_OPC_Set;
		MM2VIS.bBusAlive := OPC2MM.bBusAlive;
		MM2VIS.bOPC_Dem := OPC2MM.bOPC_Dem;
	END_IF

	IF EDGEPOS(VIS2MM.iSelExtP_OPC_Set = 0) OR EDGEPOS(VIS2MM.iSelExtP_OPC_Set = 1) OR EDGEPOS(VIS2MM.iSelExtP_OPC_Set = 2) THEN //Beim Umschalten der externen Leistungvorgabe,
		MM2VIS.bOPC_Dem := FALSE;																								 //wird der Motor abgefordert, falls die OPC-Verbidnung nicht vorhanden ist
	END_IF

	(*PI Duration A B*)
	usDurationPI_A	:= 0;
	usDurationPI_B	:= 0;
	FOR i:= 1 TO 5 DO
		usDurationPI_A	:= usDurationPI_A + IN_DI.tPIopenL[i].duration 	+ IN_DI.tPIopenH[i].duration;
		usDurationPI_B	:= usDurationPI_B + IN_DI.tPIopenL[i+5].duration + IN_DI.tPIopenH[i+5].duration;
	END_FOR

	(*Ext CAT temp setpoint*)
	MM2VIS.rCAT_TempSet 				:=	IN_DI.rCAT_TempSet;
	MM2VIS.bExtCAT_TempStatus_Active	:=	OUT_DI.bExtCAT_Temp_Active;
	MM2VIS.rExtCAT_TempSet				:=	OUT_DI.rExtCAT_TempSet;

END_PROGRAM
```

#### Gnl_ME.var
```iecst
VAR
	i : INT;
END_VAR
```

### Program Logical/DataInterface/OpcAG (IEC) - OPC Var for Testbench

#### OpcAG.st
```iecst
(*******************************************************************************
OpcAG	 Variables read or write to Testbench

This code is confidential AND proprietary to the INNIO Company.
It may NOT be used in any form, or reproduced in any manner, without the express
written permission of the INNIO Company.
Copyright, INNIO Company, 2022

- list addidtional customized IO channels

Customized modifications: -
------------------------

History:
-------
V1.00.0	14.09.2022		Vockenberger	Neu erstellt
V1.01.0	25.05.2023		Vockenberger	Dauerlauftest hinzugefügt
		28.07.2023		Vockenberger	Struktur von OPC_DI geändert
		01.08.2023		Vockenberger	Parameter für Öltankskalierung hinzugefügt
		11.01.2024		Vockenberger	bEOVal_DemOpen eingefügt
V1.02.0 10.04.2024		Vockenberger	Betriebswahlschalter, Anforderungsschalter und SY-Schalter eingefügt
V1.02.1	30.10.2024		Vockenberger	ParaTB.rTB_Cust von 1..10 auf 1..19 geändert
V1.03.0	09.01.2025		Gruber St.		cleanUp after change of parameter structure

Instructions FOR use:
--------------------

Outstandings:
------------

*******************************************************************************)

PROGRAM _CYCLIC

	(**Wird von Motor-CPU geschrieben**********************)
	(**REAL**)
	rOpcAG_R[0]		:=	Para.tPreHeatWDay[0].Hour;
	rOpcAG_R[1]		:=	Para.tPreHeatWDay[0].Minute;
	rOpcAG_R[2]		:=	Para.tPreHeatWDay[1].Hour;
	rOpcAG_R[3]		:=	Para.tPreHeatWDay[1].Minute;
	rOpcAG_R[4]		:=	Para.tPreHeatWDay[2].Hour;
	rOpcAG_R[5]		:=	Para.tPreHeatWDay[2].Minute;
	rOpcAG_R[6]		:=	Para.tPreHeatWDay[3].Hour;
	rOpcAG_R[7]		:=	Para.tPreHeatWDay[3].Minute;
	rOpcAG_R[8]		:=	Para.tPreHeatWDay[4].Hour;
	rOpcAG_R[9]		:=	Para.tPreHeatWDay[4].Minute;
	rOpcAG_R[10]	:=	Para.tPreHeatWDay[5].Hour;
	rOpcAG_R[11]	:=	Para.tPreHeatWDay[5].Minute;
	rOpcAG_R[12]	:=	Para.tPreHeatWDay[6].Hour;
	rOpcAG_R[13]	:=	Para.tPreHeatWDay[6].Minute;

	rOpcAG_R[14]	:=	VIS2MM.rEndurTestTimeSet;
	rOpcAG_R[15]	:=	IN_DI.rP_Act_Filt;
	rOpcAG_R[16]	:=	INT_TO_REAL(IN_DI.iIdx_OMSS);
	rOpcAG_R[17]	:=	INT_TO_REAL(IN_DI.iIdx_RSS);
	rOpcAG_R[18]	:=	INT_TO_REAL(IN_DI.iIdx_SyOMSS);

	rOpcAG_R[19];
	rOpcAG_R[20];
	rOpcAG_R[21];
	rOpcAG_R[22];
	rOpcAG_R[23];
	rOpcAG_R[24];
	rOpcAG_R[25];
	rOpcAG_R[26];
	rOpcAG_R[27];
	rOpcAG_R[28];
	rOpcAG_R[29];

	rOpcAG_R[30];
	rOpcAG_R[31];
	rOpcAG_R[32];
	rOpcAG_R[33];
	rOpcAG_R[34];
	rOpcAG_R[35];
	rOpcAG_R[36];
	rOpcAG_R[37];
	rOpcAG_R[38];
	rOpcAG_R[39];
	rOpcAG_R[40];

	(**BOOL**)
	IF MM2VIS.bCtrlBatMon_TestRunning THEN //Damit der Visu-Button wieder auf FALSE geschrieben wird
		VIS2MM.bCtrlBatMon_ManTestStart := FALSE;
	END_IF
	bOpcAG_R[0]	:=	VIS2MM.bCtrlBatMon_ManTestStart;
	bOpcAG_R[1]	:=	IN_DI.bImp_Start;
	bOpcAG_R[2]	:=	Para.tPreHeatWDay[0].Active;
	bOpcAG_R[3]	:=	Para.tPreHeatWDay[0].Off;
	bOpcAG_R[4]	:=	Para.tPreHeatWDay[1].Active;
	bOpcAG_R[5]	:=	Para.tPreHeatWDay[1].Off;
	bOpcAG_R[6]	:=	Para.tPreHeatWDay[2].Active;
	bOpcAG_R[7]	:=	Para.tPreHeatWDay[2].Off;
	bOpcAG_R[8]	:=	Para.tPreHeatWDay[3].Active;
	bOpcAG_R[9]	:=	Para.tPreHeatWDay[3].Off;

	bOpcAG_R[10]	:=	Para.tPreHeatWDay[4].Active;
	bOpcAG_R[11]	:=	Para.tPreHeatWDay[4].Off;
	bOpcAG_R[12]	:=	Para.tPreHeatWDay[5].Active;
	bOpcAG_R[13]	:=	Para.tPreHeatWDay[5].Off;
	bOpcAG_R[14]	:=	Para.tPreHeatWDay[6].Active;
	bOpcAG_R[15]	:=	Para.tPreHeatWDay[6].Off;
	bOpcAG_R[16]	:=	Para.bPreHeatWDay_CtrActive;
	bOpcAG_R[17]	:=	VIS2MM.bEndurTestStart;
	bOpcAG_R[18]	:=	IN_DI.bEOVal_DemOpen;
	bOpcAG_R[19];

	bOpcAG_R[20];
	bOpcAG_R[21];
	bOpcAG_R[22];
	bOpcAG_R[23];
	bOpcAG_R[24];
	bOpcAG_R[25];
	bOpcAG_R[26];
	bOpcAG_R[27];
	bOpcAG_R[28];
	bOpcAG_R[29];
	bOpcAG_R[30];

	(*AuxiliariesGeneral from Testbench*)
	(**REAL**)
	MM2VIS.rU_CtrlBat1			:=	rOpcAG_W[0];
	MM2VIS.rU_CtrlBat_BatTest1	:=	rOpcAG_W[1];
	MM2VIS.rLevel_Oiltank		:=	rOpcAG_W[2];
	rEndurTestTimeMinute		:=	rOpcAG_W[3];
	rEndurTestTimeHour			:=	rOpcAG_W[4];
	rEndurTestTimeDay			:=	rOpcAG_W[5];
	rEndurTestTimeWDay			:=	rOpcAG_W[6];
	rEndurTestTimeMonth			:=	rOpcAG_W[7];
	rEndurTestTimeYear			:=	rOpcAG_W[8];
	rTB_Version					:=	rOpcAG_W[9];

	Para.rLevel_Oiltank_ScalY1	:= rOpcAG_W[10];
	Para.rLevel_Oiltank_ScalY2	:= rOpcAG_W[11];
	MM2VIS.rI_Aux				:= rOpcAG_W[12];
	MM2VIS.rP_Aux				:= rOpcAG_W[13];
	rOpcAG_W[14];
	rOpcAG_W[15];
	rOpcAG_W[16];
	rOpcAG_W[17];
	rOpcAG_W[18];
	rOpcAG_W[19];
	rOpcAG_W[20];

	(**BOOL**)
	MM2VIS.bCtrlBatMon_TestRunning	:= bOpcAG_W[0];
	MM2VIS.bReq_RefillOilPuEng		:= bOpcAG_W[1];
	MM2VIS.bDem_RefillOilPuEng		:= bOpcAG_W[2];
	MM2VIS.bPreHeatWDay_On			:= bOpcAG_W[3];
	MM2VIS.bEndurTestEnd			:= bOpcAG_W[4];
	MM2VIS.bRelAux_TB 				:= bOpcAG_W[5];
	Para.bBatCtrActive				:= bOpcAG_W[6];
	MM2VIS.bServicePageActive		:= bOpcAG_W[7];
	MM2VIS.bAirCompressor1_Run		:= bOpcAG_W[8];
	MM2VIS.bAirCompressor2_Run		:= bOpcAG_W[9];

	bOpcAG_W[10];
	bOpcAG_W[11];
	bOpcAG_W[12];
	bOpcAG_W[13];
	bOpcAG_W[14];
	bOpcAG_W[15];
	bOpcAG_W[16];
	bOpcAG_W[17];
	bOpcAG_W[18];
	bOpcAG_W[20];

END_PROGRAM
```

### Program Logical/DataInterface/OpcCU (IEC) - OPC Var for Testbench

#### OpcCU.st
```iecst
(*******************************************************************************
OpcCU	 Variables read or write to Testbench

This code is confidential AND proprietary to the INNIO Company.
It may NOT be used in any form, or reproduced in any manner, without the express
written permission of the INNIO Company.
Copyright, INNIO Company, 2025

- list addidtional customized IO channels

Customized modifications: -
------------------------

History:
-------
V1.03.0 22.01.2025	Gruber St.	new created

Instructions FOR use:
--------------------

Outstandings:
------------

*******************************************************************************)

PROGRAM _CYCLIC

	(*------------------------------------------------------------------------------
								Testbench to Engine
	-------------------------------------------------------------------------------*)

	MM2VIS.rCust_TB2Eng[0] := rOpcCU_W[0];
	MM2VIS.rCust_TB2Eng[1] := rOpcCU_W[1];
	MM2VIS.rCust_TB2Eng[2] := rOpcCU_W[2];
	MM2VIS.rCust_TB2Eng[3] := rOpcCU_W[3];
	MM2VIS.rCust_TB2Eng[4] := rOpcCU_W[4];
	MM2VIS.rCust_TB2Eng[5] := rOpcCU_W[5];
	MM2VIS.rCust_TB2Eng[6] := rOpcCU_W[6];
	MM2VIS.rCust_TB2Eng[7] := rOpcCU_W[7];
	MM2VIS.rCust_TB2Eng[8] := rOpcCU_W[8];
	MM2VIS.rCust_TB2Eng[9] := rOpcCU_W[9];
	MM2VIS.rCust_TB2Eng[10] := rOpcCU_W[10];
	MM2VIS.rCust_TB2Eng[11] := rOpcCU_W[11];
	MM2VIS.rCust_TB2Eng[12] := rOpcCU_W[12];
	MM2VIS.rCust_TB2Eng[13] := rOpcCU_W[13];
	MM2VIS.rCust_TB2Eng[14] := rOpcCU_W[14];
	MM2VIS.rCust_TB2Eng[15] := rOpcCU_W[15];
	MM2VIS.rCust_TB2Eng[16] := rOpcCU_W[16];
	MM2VIS.rCust_TB2Eng[17] := rOpcCU_W[17];
	MM2VIS.rCust_TB2Eng[18] := rOpcCU_W[18];
	MM2VIS.rCust_TB2Eng[19] := rOpcCU_W[19];
	MM2VIS.rCust_TB2Eng[20] := rOpcCU_W[20];
	MM2VIS.rCust_TB2Eng[21] := rOpcCU_W[21];
	MM2VIS.rCust_TB2Eng[22] := rOpcCU_W[22];
	MM2VIS.rCust_TB2Eng[23] := rOpcCU_W[23];
	MM2VIS.rCust_TB2Eng[24] := rOpcCU_W[24];
	MM2VIS.rCust_TB2Eng[25] := rOpcCU_W[25];
	MM2VIS.rCust_TB2Eng[26] := rOpcCU_W[26];
	MM2VIS.rCust_TB2Eng[27] := rOpcCU_W[27];
	MM2VIS.rCust_TB2Eng[28] := rOpcCU_W[28];
	MM2VIS.rCust_TB2Eng[29] := rOpcCU_W[29];
	MM2VIS.rCust_TB2Eng[30] := rOpcCU_W[30];
	MM2VIS.rCust_TB2Eng[31] := rOpcCU_W[31];
	MM2VIS.rCust_TB2Eng[32] := rOpcCU_W[32];
	MM2VIS.rCust_TB2Eng[33] := rOpcCU_W[33];
	MM2VIS.rCust_TB2Eng[34] := rOpcCU_W[34];
	MM2VIS.rCust_TB2Eng[35] := rOpcCU_W[35];
	MM2VIS.rCust_TB2Eng[36] := rOpcCU_W[36];
	MM2VIS.rCust_TB2Eng[37] := rOpcCU_W[37];
	MM2VIS.rCust_TB2Eng[38] := rOpcCU_W[38];
	MM2VIS.rCust_TB2Eng[39] := rOpcCU_W[39];
	MM2VIS.rCust_TB2Eng[40] := rOpcCU_W[40];
	MM2VIS.rCust_TB2Eng[41] := rOpcCU_W[41];
	MM2VIS.rCust_TB2Eng[42] := rOpcCU_W[42];
	MM2VIS.rCust_TB2Eng[43] := rOpcCU_W[43];
	MM2VIS.rCust_TB2Eng[44] := rOpcCU_W[44];
	MM2VIS.rCust_TB2Eng[45] := rOpcCU_W[45];
	MM2VIS.rCust_TB2Eng[46] := rOpcCU_W[46];
	MM2VIS.rCust_TB2Eng[47] := rOpcCU_W[47];
	MM2VIS.rCust_TB2Eng[48] := rOpcCU_W[48];
	MM2VIS.rCust_TB2Eng[49] := rOpcCU_W[49];
	MM2VIS.rCust_TB2Eng[50] := rOpcCU_W[50];

	(*------------------------------------------------------------------------------
							   	Engine to Testbench
	-------------------------------------------------------------------------------*)

	rOpcCU_R[0] := VIS2MM.rCust_Eng2TB[0];
	rOpcCU_R[1] := VIS2MM.rCust_Eng2TB[1];
	rOpcCU_R[2] := VIS2MM.rCust_Eng2TB[2];
	rOpcCU_R[3] := VIS2MM.rCust_Eng2TB[3];
	rOpcCU_R[4] := VIS2MM.rCust_Eng2TB[4];
	rOpcCU_R[5] := VIS2MM.rCust_Eng2TB[5];
	rOpcCU_R[6] := VIS2MM.rCust_Eng2TB[6];
	rOpcCU_R[7] := VIS2MM.rCust_Eng2TB[7];
	rOpcCU_R[8] := VIS2MM.rCust_Eng2TB[8];
	rOpcCU_R[9] := VIS2MM.rCust_Eng2TB[9];
	rOpcCU_R[10] := VIS2MM.rCust_Eng2TB[10];
	rOpcCU_R[11] := VIS2MM.rCust_Eng2TB[11];
	rOpcCU_R[12] := VIS2MM.rCust_Eng2TB[12];
	rOpcCU_R[13] := VIS2MM.rCust_Eng2TB[13];
	rOpcCU_R[14] := VIS2MM.rCust_Eng2TB[14];
	rOpcCU_R[15] := VIS2MM.rCust_Eng2TB[15];
	rOpcCU_R[16] := VIS2MM.rCust_Eng2TB[16];
	rOpcCU_R[17] := VIS2MM.rCust_Eng2TB[17];
	rOpcCU_R[18] := VIS2MM.rCust_Eng2TB[18];
	rOpcCU_R[19] := VIS2MM.rCust_Eng2TB[19];
	rOpcCU_R[20] := VIS2MM.rCust_Eng2TB[20];
	rOpcCU_R[21] := VIS2MM.rCust_Eng2TB[21];
	rOpcCU_R[22] := VIS2MM.rCust_Eng2TB[22];
	rOpcCU_R[23] := VIS2MM.rCust_Eng2TB[23];
	rOpcCU_R[24] := VIS2MM.rCust_Eng2TB[24];
	rOpcCU_R[25] := VIS2MM.rCust_Eng2TB[25];
	rOpcCU_R[26] := VIS2MM.rCust_Eng2TB[26];
	rOpcCU_R[27] := VIS2MM.rCust_Eng2TB[27];
	rOpcCU_R[28] := VIS2MM.rCust_Eng2TB[28];
	rOpcCU_R[29] := VIS2MM.rCust_Eng2TB[29];
	rOpcCU_R[30] := VIS2MM.rCust_Eng2TB[30];
	rOpcCU_R[31] := VIS2MM.rCust_Eng2TB[31];
	rOpcCU_R[32] := VIS2MM.rCust_Eng2TB[32];
	rOpcCU_R[33] := VIS2MM.rCust_Eng2TB[33];
	rOpcCU_R[34] := VIS2MM.rCust_Eng2TB[34];
	rOpcCU_R[35] := VIS2MM.rCust_Eng2TB[35];
	rOpcCU_R[36] := VIS2MM.rCust_Eng2TB[36];
	rOpcCU_R[37] := VIS2MM.rCust_Eng2TB[37];
	rOpcCU_R[38] := VIS2MM.rCust_Eng2TB[38];
	rOpcCU_R[39] := VIS2MM.rCust_Eng2TB[39];
	rOpcCU_R[40] := VIS2MM.rCust_Eng2TB[40];
	rOpcCU_R[41] := VIS2MM.rCust_Eng2TB[41];
	rOpcCU_R[42] := VIS2MM.rCust_Eng2TB[42];
	rOpcCU_R[43] := VIS2MM.rCust_Eng2TB[43];
	rOpcCU_R[44] := VIS2MM.rCust_Eng2TB[44];
	rOpcCU_R[45] := VIS2MM.rCust_Eng2TB[45];
	rOpcCU_R[46] := VIS2MM.rCust_Eng2TB[46];
	rOpcCU_R[47] := VIS2MM.rCust_Eng2TB[47];
	rOpcCU_R[48] := VIS2MM.rCust_Eng2TB[48];
	rOpcCU_R[49] := VIS2MM.rCust_Eng2TB[49];
	rOpcCU_R[50] := VIS2MM.rCust_Eng2TB[50];

END_PROGRAM
```

### Program Logical/DataInterface/OpcEX (IEC) - OPC Var for Testbench

#### OpcEX.st
```iecst
(*******************************************************************************
OpcEX	 Variables read or write to Testbench

This code is confidential AND proprietary to the INNIO Company.
It may NOT be used in any form, or reproduced in any manner, without the express
written permission of the INNIO Company.
Copyright, INNIO Company, 2022

- list addidtional customized IO channels

Customized modifications: -
------------------------

History:
-------
V1.00.0	14.09.2022		Vockenberger	Neu erstellt
V1.01.0	28.07.2023		Vockenberger	Struktur von OPC_DI geändert
V1.02.0	20.03.2024		Vockenberger	2. Abgasgegendruckklappe hinzugefügt
V1.03.0	09.01.2025		Gruber St.		cleanUp after change of parameter structure

Instructions FOR use:
--------------------

Outstandings:
------------

*******************************************************************************)

PROGRAM _CYCLIC

	(**Wird von Motor-CPU geschrieben**********************)
	(**REAL**)

	rOpcEX_R[0]		:= VIS2MM.tCtr_EG_Flap_In.Y_man;
	rOpcEX_R[1]		:= VIS2MM.tCtr_EG_Flap_In.X_min;
	rOpcEX_R[2]		:= VIS2MM.tCtr_EG_Flap_In.X_max;
	rOpcEX_R[3]		:= INT_TO_REAL(VIS2MM.tCtr_EG_Flap_In.Tune_quality);
	rOpcEX_R[4]		:= VIS2MM.rOp_ExhFlap;
	rOpcEX_R[5]		:= VIS2MM.rMan_DPF_EgFlap_Set;
	rOpcEX_R[6]		:= VIS2MM.rMan_DPF_ByFlap_Set;
	rOpcEX_R[7]		:= VIS2MM.rMan_SRC_EgFlap_Set;
	rOpcEX_R[8]		:= VIS2MM.rMan_SRC_ByFlap_Set;
	rOpcEX_R[9]		:= VIS2MM.rCtr_EG_Flap;
	rOpcEX_R[10]	:= VIS2MM.rMan_EG_Flap_Set;

	rOpcEX_R[11];
	rOpcEX_R[12];
	rOpcEX_R[13];
	rOpcEX_R[14];
	rOpcEX_R[15];
	rOpcEX_R[16];
	rOpcEX_R[17];
	rOpcEX_R[18];
	rOpcEX_R[19];
	rOpcEX_R[20];

	rOpcEX_R[21];
	rOpcEX_R[22];
	rOpcEX_R[23];
	rOpcEX_R[24];
	rOpcEX_R[25];
	rOpcEX_R[26];
	rOpcEX_R[27];
	rOpcEX_R[28];
	rOpcEX_R[29];
	rOpcEX_R[30];

	(**BOOL**)
	bOpcEX_R[0]	:= VIS2MM.tCtr_EG_Flap_In.Y_man_Active;
	bOpcEX_R[1]	:= VIS2MM.tCtr_EG_Flap_In.W_ext_Active;
	bOpcEX_R[2]	:= VIS2MM.tCtr_EG_Flap_In.Tune_PI;
	bOpcEX_R[3]	:= VIS2MM.tCtr_EG_Flap_In.Tune_PID;
	bOpcEX_R[4]	:= VIS2MM.tCtr_EG_Flap_In.Tune_start;
	bOpcEX_R[5]	:= VIS2MM.tCtr_EG_Flap_In.Tune_stop;
	bOpcEX_R[6]	:= VIS2MM.tCtr_EG_Flap_In.Tune_takeover;
	bOpcEX_R[7];
	bOpcEX_R[8];
	bOpcEX_R[9];
	bOpcEX_R[10];

	bOpcEX_R[11];
	bOpcEX_R[12];
	bOpcEX_R[13];
	bOpcEX_R[14];
	bOpcEX_R[15];
	bOpcEX_R[16];
	bOpcEX_R[17];
	bOpcEX_R[18];
	bOpcEX_R[19];
	bOpcEX_R[20];

	(*Exhaust from Testbench*)
	(**REAL**)
	MM2VIS.rPosAct_SCR_EG_Flap	:=	rOpcEX_W[0];
	MM2VIS.rPosAct_SCR_By_Flap	:=	rOpcEX_W[1];
	MM2VIS.rPosAct_DPF_EG_Flap	:=	rOpcEX_W[2];
	MM2VIS.rPosAct_DPF_By_Flap	:=	rOpcEX_W[3];
	MM2VIS.rPr_EG_Deflag		:=	rOpcEX_W[4];
	MM2VIS.rCtr_SCR_EG_Flap_Set	:=	rOpcEX_W[5];
	MM2VIS.rCtr_SCR_By_Flap_Set	:=	rOpcEX_W[6];
	MM2VIS.rCtr_DPF_EG_Flap_Set	:=	rOpcEX_W[7];
	MM2VIS.rCtr_DPF_By_Flap_Set	:=	rOpcEX_W[8];
	MM2VIS.rCtr_EG_Flap			:=	rOpcEX_W[9];
	MM2VIS.rT_EG_PrReliefVa1	:=	rOpcEX_W[10];
	MM2VIS.rT_EG_PrReliefVa2	:=	rOpcEX_W[11];
	MM2VIS.rPr_EG_Deflag_Fast	:=	rOpcEX_W[12];
	MM2VIS.rPr_OXIcat_In_Fast_Peak	:=	rOpcEX_W[13];
	MM2VIS.rPosAct_EG_Flap	:=	rOpcEX_W[14];
	MM2VIS.rCtr_EG_Flap_Set	:=	rOpcEX_W[15];
	MM2VIS.rPosAct_EG_Flap2	:=	rOpcEX_W[16];
	rOpcEX_W[17];
	rOpcEX_W[18];
	rOpcEX_W[19];

	rOpcEX_W[20];
	rOpcEX_W[21];
	rOpcEX_W[22];
	rOpcEX_W[23];
	rOpcEX_W[24];
	rOpcEX_W[25];
	rOpcEX_W[26];
	rOpcEX_W[27];
	rOpcEX_W[28];
	rOpcEX_W[29];
	rOpcEX_W[30];

	(**BOOL**)
	MM2VIS.bSCR_Exh_Flap_O	:=	bOpcEX_W[0];
	MM2VIS.bSCR_Exh_Flap_C	:=	bOpcEX_W[1];
	MM2VIS.bSCR_By_Flap_O	:=	bOpcEX_W[2];
	MM2VIS.bSCR_By_Flap_C	:=	bOpcEX_W[3];
	MM2VIS.bDPF_Exh_Flap_O	:=	bOpcEX_W[4];
	MM2VIS.bDPF_Exh_Flap_C	:=	bOpcEX_W[5];
	MM2VIS.bDPF_By_Flap_O	:=	bOpcEX_W[6];
	MM2VIS.bDPF_By_Flap_C	:=	bOpcEX_W[7];

	Para.bEG_SRC_DPF_Active		:=	bOpcEX_W[8];
	Para.bEG_Flap2_Active		:=	bOpcEX_W[9];
	Para.bPr_EG_DeflagActive	:=	bOpcEX_W[10];
	Para.bPr_EG_DeflagFastActive	:=	bOpcEX_W[11];
	Para.bT_EG_PrReliefVa_Active	:=	bOpcEX_W[12];

	bOpcEX_W[13];
	bOpcEX_W[14];
	bOpcEX_W[15];
	bOpcEX_W[16];
	bOpcEX_W[17];
	bOpcEX_W[18];
	bOpcEX_W[19];
	bOpcEX_W[20];

END_PROGRAM
```

### Program Logical/DataInterface/OpcGT (IEC) - OPC Var for Testbench

#### OpcGT.st
```iecst
(*******************************************************************************
OpcGT	 Variables read or write to Testbench

This code is confidential AND proprietary to the INNIO Company.
It may NOT be used in any form, or reproduced in any manner, without the express
written permission of the INNIO Company.
Copyright, INNIO Company, 2022

- list addidtional customized IO channels

Customized modifications: -
------------------------

History:
-------
V1.00.0	14.09.2022		Vockenberger	Neu erstellt
V1.01.0	31.05.2023		Vockenberger	Gaskompressor mit Parameterabfrage und Betriebsstundenzähler mit Wartungsanforderung
										Parameterabfrage für Gaszähler Sensycal und Berechnet erstellt
										Parameter fürs Gasmischen eingefügt
		11.07.2023		Gruber St.		Parameter, Setpoints & Anzeigen für gastrain, clean up
		28.07.2023		Vockenberger	Struktur von OPC_DI geändert
		09.01.2024		Gruber St.		added blockage bits for mixgas & special gas
		04.03.2024		Gruber St.		added setpoints for admixing special gas with gas proportioning valve
V1.01.1 13.03.2024		Gruber St.		added variables and parameter for admixing H2
V1.02.0	22.04.2024		Gruber St.		increased all arrays; added parameters and signals for prechamber gascompressor & H2 content
										added counter gas consumption special gas in kg for H2
		08.05.2024		Gruber St.		added parameter for scaling gas meter NG, PG, SG
V1.02.1 16.10.2024		Vockenberger	P19 mit Erdgas Hochdruck
		07.11.2024		Gruber St.		added signals for butan operation
		15.11.2024		Gruber St.		added counter for gas consumption natural gas high pressure
V1.03.0	17.09.2024		Gruber St.		added scaling parameter for feedback gas pressure NG, PG, SG, PCG
		30.09.2024		Gruber St.		added Parameter and Status for Mixedmode
		09.01.2025		Gruber St.		cleanUp and several changes for new parameter structure
V1.03.5 15.04.2026	Vockenberger	added P06 PCG-compressor with mechanical regulating valve and tDem_PCG_Tank_FillValve, tDem_PCG_Tank_OpValve

Instructions FOR use:
--------------------

Outstandings:
------------

*******************************************************************************)

PROGRAM _CYCLIC

	(*------------------------------------------------------------------------------
										WRITE
	-------------------------------------------------------------------------------*)

	(**Wird von Motor-CPU geschrieben**********************)
	(**REAL**)
	rOpcGT_R[0]		:=	VIS2MM.tCtr_GC_1_In.Y_man;
	rOpcGT_R[1]		:=	VIS2MM.tCtr_GC_1_In.X_min;
	rOpcGT_R[2]		:=	VIS2MM.tCtr_GC_1_In.X_max;
	rOpcGT_R[3]		:=	INT_TO_REAL(VIS2MM.tCtr_GC_1_In.Tune_quality);

	rOpcGT_R[4]		:=	VIS2MM.tCtr_GC_2_In.Y_man;
	rOpcGT_R[5]		:=	VIS2MM.tCtr_GC_2_In.X_min;
	rOpcGT_R[6]		:=	VIS2MM.tCtr_GC_2_In.X_max;
	rOpcGT_R[7]		:=	INT_TO_REAL(VIS2MM.tCtr_GC_2_In.Tune_quality);

	rOpcGT_R[8]		:=	VIS2MM.tCtr_MN_MG_In.Y_man;
	rOpcGT_R[9]		:=	VIS2MM.tCtr_MN_MG_In.X_min;
	rOpcGT_R[10]	:=	VIS2MM.tCtr_MN_MG_In.X_max;
	rOpcGT_R[11]	:=	INT_TO_REAL(VIS2MM.tCtr_MN_MG_In.Tune_quality);

	rOpcGT_R[12]	:=	VIS2MM.rVol_PG_Set;
	rOpcGT_R[13]	:=	VIS2MM.rVol_SG_Set;
	rOpcGT_R[14]	:=	INT_TO_REAL(IN_DI.iIdx_SelGasTyp);

	rOpcGT_R[15]	:=	IN_DI.rGMU_Pr_FuelGas[1];
	rOpcGT_R[16]	:=	IN_DI.rGMU_T_FuelGas[1];
	rOpcGT_R[17]	:=	IN_DI.rGMU_Q_FuelGas[1];
	rOpcGT_R[18]	:=	IN_DI.rGMU_Pr_FuelGas[2];
	rOpcGT_R[19]	:=	IN_DI.rGMU_T_FuelGas[2];
	rOpcGT_R[20]	:=	IN_DI.rGMU_Q_FuelGas[2];
	rOpcGT_R[21]	:=	IN_DI.rGMU_Pr_FuelGas[3];
	rOpcGT_R[22]	:=	IN_DI.rGMU_T_FuelGas[3];
	rOpcGT_R[23]	:=	IN_DI.rGMU_Q_FuelGas[3];

	rOpcGT_R[24]	:=	Para.tCtr_GC_1.W_set;
	rOpcGT_R[25]	:=	Para.tCtr_GC_2.W_set;
	rOpcGT_R[26]	:=	Para.tCtr_MN_MG.W_set;
	rOpcGT_R[27]	:=	Para.rSel_LSCS_GV;
	rOpcGT_R[28]	:=	Para.rLSCS_GV_Set;
	rOpcGT_R[29]	:=	Para.rSel_LSCS_MV;
	rOpcGT_R[30]	:=	Para.rLSCS_MV_Set;
	rOpcGT_R[31]	:=	Para.rCnt_CompOpHoursW;

	rOpcGT_R[32]	:=	VIS2MM.rCtr_PG_CompSet;
	rOpcGT_R[33]	:=	VIS2MM.rCtr_GasTempSet;
	rOpcGT_R[34]	:=	IN_DI.rQg_set_A;
	rOpcGT_R[35]	:=	IN_DI.rQg_set_B;
	rOpcGT_R[36]	:=	IN_DI.rZDKappaPE;

	(* ----------------------------------------------------------------------------*)
	(**BOOL*)
	bOpcGT_R[0]	:=	VIS2MM.bDemDataMan_GC;
	TON_DemDataMan_GC(IN:=VIS2MM.bDemDataMan_GC, PT:=T#500ms);
	IF TON_DemDataMan_GC.Q THEN //Damit der Visu-Button wieder auf FALSE geschrieben wird
		VIS2MM.bDemDataMan_GC := FALSE;
	END_IF

	bOpcGT_R[1] := VIS2MM.bCtr_MN_MG_active;
	bOpcGT_R[2] := VIS2MM.bCtr_MN_MG_off;
	bOpcGT_R[3] := VIS2MM.bVolPG_Man;
	bOpcGT_R[4]	:= IN_DI.bGV1_Open;
	bOpcGT_R[5]	:= IN_DI.bGV2_Open;
	bOpcGT_R[6]	:= Para.bIncl_SG_Calc;
	bOpcGT_R[7]	:= Para.bSend_Cv2Eng;
	bOpcGT_R[8]	:= REAL_TO_BOOL(Para.rTB_Cust[14]);	(*Butan Operation active (ParaGT.bBG_Operation)*)
	bOpcGT_R[9]	:= OUT_DI.bCompOpHoursWarning;

	bOpcGT_R[10]	:= VIS2MM.bSel_PG_Comp;
	bOpcGT_R[11]	:= VIS2MM.bSel_PG_TraceHeat;
	bOpcGT_R[12]	:= VIS2MM.bSel_PG_TraceHeat_TimeCtr;
	bOpcGT_R[13]	:= IN_DI.bSA_PI_Active;

	(*------------------------------------------------------------------------------
										READ
	-------------------------------------------------------------------------------*)

	(*Gastrain from Testbench*)
	MM2VIS.rVol_GT_NG		:=	rOpcGT_W[0];
	MM2VIS.rVol_GT_PG		:=	rOpcGT_W[1];
	MM2VIS.rVol_GT_SG		:=	rOpcGT_W[2];
	MM2VIS.rMFC_Act_PG		:=	rOpcGT_W[3];
	MM2VIS.rMFC_Act_SG		:=	rOpcGT_W[4];
	MM2VIS.rPosAct_LSCS_GV	:=	rOpcGT_W[5];
	MM2VIS.rPosAct_LSCS_MV	:=	rOpcGT_W[6];
	MM2VIS.rPr_GT_NG		:=	rOpcGT_W[7];
	MM2VIS.rPr_GT_PG		:=	rOpcGT_W[8];
	MM2VIS.rPr_GT_SG		:=	rOpcGT_W[9];

	MM2VIS.rPr_PCG_Tank		:=	rOpcGT_W[10];
	MM2VIS.rT_GT_NG			:=	rOpcGT_W[11];
	MM2VIS.rT_GT_PG			:=	rOpcGT_W[12];
	MM2VIS.rT_GT_SG			:=	rOpcGT_W[13];
	MM2VIS.rCtr_MFC_PG		:=	rOpcGT_W[14];
	MM2VIS.rCtr_MFC_SG		:=	rOpcGT_W[15];
	MM2VIS.rCtr_By1_GComp	:=	rOpcGT_W[16];
	MM2VIS.rCtr_By2_GComp	:=	rOpcGT_W[17];
	MM2VIS.rCtr_LSCS_GV		:=	rOpcGT_W[18];
	MM2VIS.rCtr_LSCS_MV		:=	rOpcGT_W[19];

	MM2VIS.rAct_LSCS_MV_Calc	:=	rOpcGT_W[20];
	MM2VIS.rAct_LSCS_GV_Calc	:=	rOpcGT_W[21];
	MM2VIS.rLSCS_Diff			:=	rOpcGT_W[22];
	MM2VIS.rCtr_MFC_PG_Set		:=	rOpcGT_W[23];
	MM2VIS.rCtr_MFC_SG_Set		:=	rOpcGT_W[24];
	MM2VIS.rCnt_Gas_M3			:=	rOpcGT_W[25];
	MM2VIS.rCnt_OpHours			:=	rOpcGT_W[26];
	MM2VIS.rCnt_Starts			:=	rOpcGT_W[27];
	MM2VIS.rCnt_CompOpHours		:=	rOpcGT_W[28];
	rOpcGT_W[29];

	MM2VIS.tGasconsumMonth[0].ConsumNG	:=	rOpcGT_W[30];
	MM2VIS.tGasconsumMonth[1].ConsumNG	:=	rOpcGT_W[31];
	MM2VIS.tGasconsumMonth[2].ConsumNG	:=	rOpcGT_W[32];
	MM2VIS.tGasconsumMonth[3].ConsumNG	:=	rOpcGT_W[33];
	MM2VIS.tGasconsumMonth[4].ConsumNG	:=	rOpcGT_W[34];
	MM2VIS.tGasconsumMonth[5].ConsumNG	:=	rOpcGT_W[35];
	MM2VIS.tGasconsumMonth[6].ConsumNG	:=	rOpcGT_W[36];
	MM2VIS.tGasconsumMonth[7].ConsumNG	:=	rOpcGT_W[37];
	MM2VIS.tGasconsumMonth[8].ConsumNG	:=	rOpcGT_W[38];
	MM2VIS.tGasconsumMonth[9].ConsumNG	:=	rOpcGT_W[39];
	MM2VIS.tGasconsumMonth[10].ConsumNG	:=	rOpcGT_W[40];
	MM2VIS.tGasconsumMonth[11].ConsumNG	:=	rOpcGT_W[41];
	MM2VIS.tGasconsumMonth[12].ConsumNG	:=	rOpcGT_W[42];

	MM2VIS.tGasconsumMonth[0].ConsumPG	:=	rOpcGT_W[43];
	MM2VIS.tGasconsumMonth[1].ConsumPG	:=	rOpcGT_W[44];
	MM2VIS.tGasconsumMonth[2].ConsumPG	:=	rOpcGT_W[45];
	MM2VIS.tGasconsumMonth[3].ConsumPG	:=	rOpcGT_W[46];
	MM2VIS.tGasconsumMonth[4].ConsumPG	:=	rOpcGT_W[47];
	MM2VIS.tGasconsumMonth[5].ConsumPG	:=	rOpcGT_W[48];
	MM2VIS.tGasconsumMonth[6].ConsumPG	:=	rOpcGT_W[49];
	MM2VIS.tGasconsumMonth[7].ConsumPG	:=	rOpcGT_W[50];
	MM2VIS.tGasconsumMonth[8].ConsumPG	:=	rOpcGT_W[51];
	MM2VIS.tGasconsumMonth[9].ConsumPG	:=	rOpcGT_W[52];
	MM2VIS.tGasconsumMonth[10].ConsumPG	:=	rOpcGT_W[53];
	MM2VIS.tGasconsumMonth[11].ConsumPG	:=	rOpcGT_W[54];
	MM2VIS.tGasconsumMonth[12].ConsumPG	:=	rOpcGT_W[55];

	MM2VIS.tGasconsumMonth[0].OpHours	:=	rOpcGT_W[56];
	MM2VIS.tGasconsumMonth[1].OpHours	:=	rOpcGT_W[57];
	MM2VIS.tGasconsumMonth[2].OpHours	:=	rOpcGT_W[58];
	MM2VIS.tGasconsumMonth[3].OpHours	:=	rOpcGT_W[59];
	MM2VIS.tGasconsumMonth[4].OpHours	:=	rOpcGT_W[60];
	MM2VIS.tGasconsumMonth[5].OpHours	:=	rOpcGT_W[61];
	MM2VIS.tGasconsumMonth[6].OpHours	:=	rOpcGT_W[62];
	MM2VIS.tGasconsumMonth[7].OpHours	:=	rOpcGT_W[63];
	MM2VIS.tGasconsumMonth[8].OpHours	:=	rOpcGT_W[64];
	MM2VIS.tGasconsumMonth[9].OpHours	:=	rOpcGT_W[65];
	MM2VIS.tGasconsumMonth[10].OpHours	:=	rOpcGT_W[66];
	MM2VIS.tGasconsumMonth[11].OpHours	:=	rOpcGT_W[67];
	MM2VIS.tGasconsumMonth[12].OpHours	:=	rOpcGT_W[68];

	MM2VIS.tGasconsumMonth[0].P_WorkAct	:=	rOpcGT_W[69];
	MM2VIS.tGasconsumMonth[1].P_WorkAct	:=	rOpcGT_W[70];
	MM2VIS.tGasconsumMonth[2].P_WorkAct	:=	rOpcGT_W[71];
	MM2VIS.tGasconsumMonth[3].P_WorkAct	:=	rOpcGT_W[72];
	MM2VIS.tGasconsumMonth[4].P_WorkAct	:=	rOpcGT_W[73];
	MM2VIS.tGasconsumMonth[5].P_WorkAct	:=	rOpcGT_W[74];
	MM2VIS.tGasconsumMonth[6].P_WorkAct	:=	rOpcGT_W[75];
	MM2VIS.tGasconsumMonth[7].P_WorkAct	:=	rOpcGT_W[76];
	MM2VIS.tGasconsumMonth[8].P_WorkAct	:=	rOpcGT_W[77];
	MM2VIS.tGasconsumMonth[9].P_WorkAct	:=	rOpcGT_W[78];
	MM2VIS.tGasconsumMonth[10].P_WorkAct	:=	rOpcGT_W[79];
	MM2VIS.tGasconsumMonth[11].P_WorkAct	:=	rOpcGT_W[80];
	MM2VIS.tGasconsumMonth[12].P_WorkAct	:=	rOpcGT_W[81];

	MM2VIS.tGasconsumYear[0].Year	:=	rOpcGT_W[82];
	MM2VIS.tGasconsumYear[1].Year	:=	rOpcGT_W[83];
	MM2VIS.tGasconsumYear[2].Year	:=	rOpcGT_W[84];
	MM2VIS.tGasconsumYear[3].Year	:=	rOpcGT_W[85];
	MM2VIS.tGasconsumYear[4].Year	:=	rOpcGT_W[86];
	MM2VIS.tGasconsumYear[5].Year	:=	rOpcGT_W[87];
	MM2VIS.tGasconsumYear[6].Year	:=	rOpcGT_W[88];
	MM2VIS.tGasconsumYear[7].Year	:=	rOpcGT_W[89];
	MM2VIS.tGasconsumYear[8].Year	:=	rOpcGT_W[90];
	MM2VIS.tGasconsumYear[9].Year	:=	rOpcGT_W[91];

	MM2VIS.tGasconsumYear[0].ConsumNG	:=	rOpcGT_W[92];
	MM2VIS.tGasconsumYear[1].ConsumNG	:=	rOpcGT_W[93];
	MM2VIS.tGasconsumYear[2].ConsumNG	:=	rOpcGT_W[94];
	MM2VIS.tGasconsumYear[3].ConsumNG	:=	rOpcGT_W[95];
	MM2VIS.tGasconsumYear[4].ConsumNG	:=	rOpcGT_W[96];
	MM2VIS.tGasconsumYear[5].ConsumNG	:=	rOpcGT_W[97];
	MM2VIS.tGasconsumYear[6].ConsumNG	:=	rOpcGT_W[98];
	MM2VIS.tGasconsumYear[7].ConsumNG	:=	rOpcGT_W[99];
	MM2VIS.tGasconsumYear[8].ConsumNG	:=	rOpcGT_W[100];
	MM2VIS.tGasconsumYear[9].ConsumNG	:=	rOpcGT_W[101];

	MM2VIS.tGasconsumYear[0].ConsumPG	:=	rOpcGT_W[102];
	MM2VIS.tGasconsumYear[1].ConsumPG	:=	rOpcGT_W[103];
	MM2VIS.tGasconsumYear[2].ConsumPG	:=	rOpcGT_W[104];
	MM2VIS.tGasconsumYear[3].ConsumPG	:=	rOpcGT_W[105];
	MM2VIS.tGasconsumYear[4].ConsumPG	:=	rOpcGT_W[106];
	MM2VIS.tGasconsumYear[5].ConsumPG	:=	rOpcGT_W[107];
	MM2VIS.tGasconsumYear[6].ConsumPG	:=	rOpcGT_W[108];
	MM2VIS.tGasconsumYear[7].ConsumPG	:=	rOpcGT_W[109];
	MM2VIS.tGasconsumYear[8].ConsumPG	:=	rOpcGT_W[110];
	MM2VIS.tGasconsumYear[9].ConsumPG	:=	rOpcGT_W[111];

	MM2VIS.tGasconsumYear[0].P_WorkAct	:=	rOpcGT_W[112];
	MM2VIS.tGasconsumYear[1].P_WorkAct	:=	rOpcGT_W[113];
	MM2VIS.tGasconsumYear[2].P_WorkAct	:=	rOpcGT_W[114];
	MM2VIS.tGasconsumYear[3].P_WorkAct	:=	rOpcGT_W[115];
	MM2VIS.tGasconsumYear[4].P_WorkAct	:=	rOpcGT_W[116];
	MM2VIS.tGasconsumYear[5].P_WorkAct	:=	rOpcGT_W[117];
	MM2VIS.tGasconsumYear[6].P_WorkAct	:=	rOpcGT_W[118];
	MM2VIS.tGasconsumYear[7].P_WorkAct	:=	rOpcGT_W[119];
	MM2VIS.tGasconsumYear[8].P_WorkAct	:=	rOpcGT_W[120];
	MM2VIS.tGasconsumYear[9].P_WorkAct	:=	rOpcGT_W[121];

	MM2VIS.tGasconsumMonth[0].ConsumSG	:=	rOpcGT_W[122];
	MM2VIS.tGasconsumMonth[1].ConsumSG	:=	rOpcGT_W[123];
	MM2VIS.tGasconsumMonth[2].ConsumSG	:=	rOpcGT_W[124];
	MM2VIS.tGasconsumMonth[3].ConsumSG	:=	rOpcGT_W[125];
	MM2VIS.tGasconsumMonth[4].ConsumSG	:=	rOpcGT_W[126];
	MM2VIS.tGasconsumMonth[5].ConsumSG	:=	rOpcGT_W[127];
	MM2VIS.tGasconsumMonth[6].ConsumSG	:=	rOpcGT_W[128];
	MM2VIS.tGasconsumMonth[7].ConsumSG	:=	rOpcGT_W[129];
	MM2VIS.tGasconsumMonth[8].ConsumSG	:=	rOpcGT_W[130];
	MM2VIS.tGasconsumMonth[9].ConsumSG	:=	rOpcGT_W[131];
	MM2VIS.tGasconsumMonth[10].ConsumSG	:=	rOpcGT_W[132];
	MM2VIS.tGasconsumMonth[11].ConsumSG	:=	rOpcGT_W[133];
	MM2VIS.tGasconsumMonth[12].ConsumSG	:=	rOpcGT_W[134];

	MM2VIS.tGasconsumYear[0].ConsumSG	:=	rOpcGT_W[135];
	MM2VIS.tGasconsumYear[1].ConsumSG	:=	rOpcGT_W[136];
	MM2VIS.tGasconsumYear[2].ConsumSG	:=	rOpcGT_W[137];
	MM2VIS.tGasconsumYear[3].ConsumSG	:=	rOpcGT_W[138];
	MM2VIS.tGasconsumYear[4].ConsumSG	:=	rOpcGT_W[139];
	MM2VIS.tGasconsumYear[5].ConsumSG	:=	rOpcGT_W[140];
	MM2VIS.tGasconsumYear[6].ConsumSG	:=	rOpcGT_W[141];
	MM2VIS.tGasconsumYear[7].ConsumSG	:=	rOpcGT_W[142];
	MM2VIS.tGasconsumYear[8].ConsumSG	:=	rOpcGT_W[143];
	MM2VIS.tGasconsumYear[9].ConsumSG	:=	rOpcGT_W[144];

	MM2VIS.tGasconsumYear[0].OpHours	:=	rOpcGT_W[145];
	MM2VIS.tGasconsumYear[1].OpHours	:=	rOpcGT_W[146];
	MM2VIS.tGasconsumYear[2].OpHours	:=	rOpcGT_W[147];
	MM2VIS.tGasconsumYear[3].OpHours	:=	rOpcGT_W[148];
	MM2VIS.tGasconsumYear[4].OpHours	:=	rOpcGT_W[149];
	MM2VIS.tGasconsumYear[5].OpHours	:=	rOpcGT_W[150];
	MM2VIS.tGasconsumYear[6].OpHours	:=	rOpcGT_W[151];
	MM2VIS.tGasconsumYear[7].OpHours	:=	rOpcGT_W[152];
	MM2VIS.tGasconsumYear[8].OpHours	:=	rOpcGT_W[153];
	MM2VIS.tGasconsumYear[9].OpHours	:=	rOpcGT_W[154];

	MM2VIS.rNG_C3H8 := rOpcGT_W[155];
	MM2VIS.rNG_C4H10 := rOpcGT_W[156];
	MM2VIS.rNG_C5H12 := rOpcGT_W[157];
	IF MM2VIS.bMN_Cal_Status = TRUE THEN
		MM2VIS.rMN_MG := rOpcGT_W[158];
		MM2VIS.rMN_NG := rOpcGT_W[159];
	ELSE
		MM2VIS.rMN_MG := 0;
		MM2VIS.rMN_NG := 0;
	END_IF
	MM2VIS.rCtr_MN_MG_Out_Y := rOpcGT_W[160];
	MM2VIS.rNG_C6H14 := rOpcGT_W[161];
	MM2VIS.rNG_N2 := rOpcGT_W[162];
	MM2VIS.rNG_CH4 := rOpcGT_W[163];
	MM2VIS.rNG_CO2 := rOpcGT_W[164];
	MM2VIS.rNG_C2H6 := rOpcGT_W[165];

	MM2VIS.rPG_C3H8 := rOpcGT_W[166];
	MM2VIS.rPG_C4H10 := rOpcGT_W[167];
	MM2VIS.rPG_C5H12 := rOpcGT_W[168];
	MM2VIS.rSum_GT_NG_Norm := rOpcGT_W[169];
	IF MM2VIS.bMN_Cal_Status = TRUE THEN
		MM2VIS.rMN_PG := rOpcGT_W[170];
	ELSE
		MM2VIS.rMN_PG := 0;
	END_IF
	rOpcGT_W[171];
	MM2VIS.rPG_C6H14 := rOpcGT_W[172];
	MM2VIS.rPG_N2 := rOpcGT_W[173];
	MM2VIS.rPG_CH4 := rOpcGT_W[174];
	MM2VIS.rPG_CO2 := rOpcGT_W[175];
	MM2VIS.rPG_C2H6 := rOpcGT_W[176];

	rGC_CurrentMonth := rOpcGT_W[177];
	rGC_CurrentDay := rOpcGT_W[178];
	rGC_CurrentYear := rOpcGT_W[179];
	rGC_CurrentHour := rOpcGT_W[180];
	rGC_CurrentMinute := rOpcGT_W[181];
	rGC_SampleMonth := rOpcGT_W[182];
	rGC_SampleDay := rOpcGT_W[183];
	rGC_SampleYear := rOpcGT_W[184];
	rGC_SampleHour := rOpcGT_W[185];
	rGC_SampleMinute := rOpcGT_W[186];

	MM2VIS.rGT_CH4_TB := rOpcGT_W[187];
	MM2VIS.rGT_CV_TB := rOpcGT_W[188];
	MM2VIS.rVol_PG := rOpcGT_W[189];
	MM2VIS.rVol_SG := rOpcGT_W[190];
	MM2VIS.rVol_NG := rOpcGT_W[191];
	MM2VIS.rGT_RatioMix_Set	:= rOpcGT_W[192];
	rGT_RatioAdd := rOpcGT_W[193];
	rH2_Set := rOpcGT_W[194];
	rH2_Act_Calc := rOpcGT_W[195];
	rH2_Act_Cube := rOpcGT_W[196];
	MM2VIS.rT_PCGAfComp := rOpcGT_W[197];
	MM2VIS.rT_PCGAfCooler := rOpcGT_W[198];

	MM2VIS.tGasconsumMonth[0].ConsumH2	:=	rOpcGT_W[199];
	MM2VIS.tGasconsumMonth[1].ConsumH2	:=	rOpcGT_W[200];
	MM2VIS.tGasconsumMonth[2].ConsumH2	:=	rOpcGT_W[201];
	MM2VIS.tGasconsumMonth[3].ConsumH2	:=	rOpcGT_W[202];
	MM2VIS.tGasconsumMonth[4].ConsumH2	:=	rOpcGT_W[203];
	MM2VIS.tGasconsumMonth[5].ConsumH2	:=	rOpcGT_W[204];
	MM2VIS.tGasconsumMonth[6].ConsumH2	:=	rOpcGT_W[205];
	MM2VIS.tGasconsumMonth[7].ConsumH2	:=	rOpcGT_W[206];
	MM2VIS.tGasconsumMonth[8].ConsumH2	:=	rOpcGT_W[207];
	MM2VIS.tGasconsumMonth[9].ConsumH2	:=	rOpcGT_W[208];
	MM2VIS.tGasconsumMonth[10].ConsumH2	:=	rOpcGT_W[209];
	MM2VIS.tGasconsumMonth[11].ConsumH2	:=	rOpcGT_W[210];
	MM2VIS.tGasconsumMonth[12].ConsumH2	:=	rOpcGT_W[211];

	MM2VIS.tGasconsumYear[0].ConsumH2	:=	rOpcGT_W[212];
	MM2VIS.tGasconsumYear[1].ConsumH2	:=	rOpcGT_W[213];
	MM2VIS.tGasconsumYear[2].ConsumH2	:=	rOpcGT_W[214];
	MM2VIS.tGasconsumYear[3].ConsumH2	:=	rOpcGT_W[215];
	MM2VIS.tGasconsumYear[4].ConsumH2	:=	rOpcGT_W[216];
	MM2VIS.tGasconsumYear[5].ConsumH2	:=	rOpcGT_W[217];
	MM2VIS.tGasconsumYear[6].ConsumH2	:=	rOpcGT_W[218];
	MM2VIS.tGasconsumYear[7].ConsumH2	:=	rOpcGT_W[219];
	MM2VIS.tGasconsumYear[8].ConsumH2	:=	rOpcGT_W[220];
	MM2VIS.tGasconsumYear[9].ConsumH2	:=	rOpcGT_W[221];

	MM2VIS.rT_GT_BG1	:=	rOpcGT_W[222];
	MM2VIS.rT_GT_BG2	:=	rOpcGT_W[223];
	MM2VIS.tGasconsumMonth[0].ConsumNG_HD	:=	rOpcGT_W[224];
	MM2VIS.tGasconsumMonth[1].ConsumNG_HD	:=	rOpcGT_W[225];
	MM2VIS.tGasconsumMonth[2].ConsumNG_HD	:=	rOpcGT_W[226];
	MM2VIS.tGasconsumMonth[3].ConsumNG_HD	:=	rOpcGT_W[227];
	MM2VIS.tGasconsumMonth[4].ConsumNG_HD	:=	rOpcGT_W[228];
	MM2VIS.tGasconsumMonth[5].ConsumNG_HD	:=	rOpcGT_W[229];
	MM2VIS.tGasconsumMonth[6].ConsumNG_HD	:=	rOpcGT_W[230];
	MM2VIS.tGasconsumMonth[7].ConsumNG_HD	:=	rOpcGT_W[231];
	MM2VIS.tGasconsumMonth[8].ConsumNG_HD	:=	rOpcGT_W[232];
	MM2VIS.tGasconsumMonth[9].ConsumNG_HD	:=	rOpcGT_W[233];
	MM2VIS.tGasconsumMonth[10].ConsumNG_HD	:=	rOpcGT_W[234];
	MM2VIS.tGasconsumMonth[11].ConsumNG_HD	:=	rOpcGT_W[235];
	MM2VIS.tGasconsumMonth[12].ConsumNG_HD	:=	rOpcGT_W[236];
	MM2VIS.tGasconsumYear[0].ConsumNG_HD	:=	rOpcGT_W[237];
	MM2VIS.tGasconsumYear[1].ConsumNG_HD	:=	rOpcGT_W[238];
	MM2VIS.tGasconsumYear[2].ConsumNG_HD	:=	rOpcGT_W[239];
	MM2VIS.tGasconsumYear[3].ConsumNG_HD	:=	rOpcGT_W[240];
	MM2VIS.tGasconsumYear[4].ConsumNG_HD	:=	rOpcGT_W[241];
	MM2VIS.tGasconsumYear[5].ConsumNG_HD	:=	rOpcGT_W[242];
	MM2VIS.tGasconsumYear[6].ConsumNG_HD	:=	rOpcGT_W[243];
	MM2VIS.tGasconsumYear[7].ConsumNG_HD	:=	rOpcGT_W[244];
	MM2VIS.tGasconsumYear[8].ConsumNG_HD	:=	rOpcGT_W[245];
	MM2VIS.tGasconsumYear[9].ConsumNG_HD	:=	rOpcGT_W[246];

	(*Parameter for vis*)
	Para.rTB_Cust[1]	:=	rOpcGT_W[247]; (*MFC Setpoint maximum propan*)
	Para.rTB_Cust[2]	:=	rOpcGT_W[248]; (*MFC Setpoint maximum special gas*)
	Para.rTB_Cust[11]	:=	rOpcGT_W[249]; (*Propan gastrain exist*)
	Para.rTB_Cust[12]	:=	rOpcGT_W[250]; (*Natural gastrain HP exist*)
	Para.rTB_Cust[13]	:=	rOpcGT_W[251]; (*Butan gastrain used*)
	Para.rT_PCGAfComp_HiHi		:=	rOpcGT_W[252];
	Para.rT_PCGAfCooler_HiHi	:=	rOpcGT_W[253];

	MM2VIS.rPr_PG_AfterComp	:=	rOpcGT_W[254];
	MM2VIS.rPr_PG_CompTank	:=	rOpcGT_W[255];
	MM2VIS.rT_PG_CompCW		:=	rOpcGT_W[256];
	MM2VIS.rT_PG_BeforeComp	:=	rOpcGT_W[257];
	MM2VIS.rT_PG_AfterComp	:=	rOpcGT_W[258];
	MM2VIS.rT_PG_Tank		:=	rOpcGT_W[259];
	MM2VIS.rCtr_PG_Comp		:=	rOpcGT_W[260];
	MM2VIS.rCtr_PG_CompCool	:=	rOpcGT_W[261];
	MM2VIS.rPr_NG_bValve	:=	rOpcGT_W[262];
	MM2VIS.rPr_PG_bValve	:=	rOpcGT_W[263];
	MM2VIS.rPr_GasAfterTempCtr	:=	rOpcGT_W[264];
	MM2VIS.rT_GasAfterTempCtr	:=	rOpcGT_W[265];
	MM2VIS.rT_GasAfterMixer		:=	rOpcGT_W[266];

	MM2VIS.rT_PCG_CW_Re		:=	rOpcGT_W[267];
	MM2VIS.rT_PCG_CW_Su		:=	rOpcGT_W[268];
	MM2VIS.rPr_PCG_CW		:=	rOpcGT_W[269];

	(* ----------------------------------------------------------------------------*)
	(**BOOL**)
	MM2VIS.bLSCS_GV_Opened		:= bOpcGT_W[0];
	MM2VIS.bLSCS_GV_Closed		:= bOpcGT_W[1];
	MM2VIS.bLSCS_MV_Opened		:= bOpcGT_W[2];
	MM2VIS.bLSCS_MV_Closed		:= bOpcGT_W[3];
	MM2VIS.bDem_FV_PCGC_NG		:= bOpcGT_W[4];
	MM2VIS.bDem_FV_PCGC_MG		:= bOpcGT_W[5];
	MM2VIS.bDem_FV_PCGC_PG		:= bOpcGT_W[6];
	MM2VIS.bDem_GV_NG			:= bOpcGT_W[7];
	MM2VIS.bDem_GV_PG			:= bOpcGT_W[8];
	MM2VIS.bDem_GV_SG			:= bOpcGT_W[9];

	MM2VIS.bDem_PCG_Val			:= bOpcGT_W[10];
	MM2VIS.bPr_PCG_GC_Dem		:= bOpcGT_W[11];
	MM2VIS.bPCG_DemReliefValve	:= bOpcGT_W[12];
	MM2VIS.bGC_Status			:= bOpcGT_W[13];
	MM2VIS.bMN_Cal_Status		:= bOpcGT_W[14];
	MM2VIS.bCtr_MN_MG_In_enable	:= bOpcGT_W[15];
	MM2VIS.bCV_Bus_Active 		:= bOpcGT_W[16];
	MM2VIS.bMixAllTrains 		:= bOpcGT_W[17];
	MM2VIS.bOptGT_RatioMix_Set 	:= bOpcGT_W[18];
	bBlock_MG_TB				:= bOpcGT_W[19];

	bBlock_SG_TB				:= bOpcGT_W[20];
	bDem_GT3					:= bOpcGT_W[21];
	MM2VIS.bDem_GV_NG_HP		:= bOpcGT_W[22];
	MM2VIS.bSel_GT_NG_HP		:= bOpcGT_W[23];
	MM2VIS.bDem_TraceHeating_BG	:= bOpcGT_W[24];
	MM2VIS.bMX_Status			:= bOpcGT_W[25];

	(*Parameter for vis*)
	Para.bSG_active			:=	bOpcGT_W[26];
	Para.bPG_MFC_Used		:=	bOpcGT_W[27];
	Para.bSG_MFC_Used		:=	bOpcGT_W[28];
	Para.bPr_GT_NG_used		:=	bOpcGT_W[29];
	Para.bPr_GT_PG_used		:=	bOpcGT_W[30];
	Para.bPr_GT_SG_used		:=	bOpcGT_W[31];
	Para.bT_GT_NG_used		:=	bOpcGT_W[32];
	Para.bT_GT_PG_used		:=	bOpcGT_W[33];
	Para.bT_GT_SG_used		:=	bOpcGT_W[34];
	Para.bFlow_GT_NG_used	:=	bOpcGT_W[35];
	Para.bFlow_GT_PG_used	:=	bOpcGT_W[36];
	Para.bFlow_GT_SG_used	:=	bOpcGT_W[37];

	Para.bPCGC_AirCooler		:=	bOpcGT_W[38];
	Para.bGasCntSensycalActive	:=	bOpcGT_W[39];
	Para.bGasCntCalcActive		:=	bOpcGT_W[40];
	Para.bGasCompActive			:=	bOpcGT_W[41];
	Para.bLSCS_GV_active		:=	bOpcGT_W[42];
	Para.bLSCS_MV_active		:=	bOpcGT_W[43];
	Para.bH2_Mode				:=	bOpcGT_W[44];
	Para.bGasFlowCtr			:=	bOpcGT_W[45];

	MM2VIS.bPG_TraceHeat_TimeCtr_On	:=	bOpcGT_W[46];
	MM2VIS.bDem_PG_TraceHeat		:=	bOpcGT_W[47];
	MM2VIS.bDem_PG_Comp_FC			:=	bOpcGT_W[48];
	MM2VIS.bDem_PG_CompValCW		:=	bOpcGT_W[49];

	MM2VIS.bDem_PCG_Tank_FillValve	:=	bOpcGT_W[50];
	MM2VIS.bDem_PCG_Tank_OpValve	:=	bOpcGT_W[51];
	MM2VIS.bPCG_Comp_CV_Mech_Active	:=	bOpcGT_W[52]; //Para from TB_Control
	MM2VIS.bPCG_MG_Valve_Inactive	:=	bOpcGT_W[53]; //Para from TB_Control
	MM2VIS.bSingle_H2_GT			:=	bOpcGT_W[54]; //Para from TB_Control
	MM2VIS.bPCG_DemValCW			:=  bOpcGT_W[55];

END_PROGRAM
```

### Program Logical/DataInterface/OpcHC (IEC) - OPC Var for Testbench
